LIN {X 0,Y 311.51,Z 741.802,A -85,B 0,C 180,E1 -15908.491,E2 -15908.491} C_VEL
LIN {X 0,Y 309.243,Z 751.676,A -85,B 0,C 180,E1 -15910.758,E2 -15910.758} C_VEL
LIN {X 0,Y 307.436,Z 759.867,A -85,B 0,C 180,E1 -15913.052,E2 -15913.052} C_VEL
LIN {X 0,Y 306.027,Z 766.633,A -85,B 0,C 180,E1 -15915.366,E2 -15915.366} C_VEL
LIN {X 0,Y 304.868,Z 772.893,A -85,B 0,C 180,E1 -15918.024,E2 -15918.024} C_VEL
LIN {X 0,Y 304.197,Z 777.728,A -85,B 0,C 180,E1 -15920.691,E2 -15920.691} C_VEL
LIN {X 0,Y 303.83,Z 781.267,A -85,B 0,C 180,E1 -15923.357,E2 -15923.357} C_VEL
LIN {X 0,Y 303.672,Z 783.591,A -85,B 0,C 180,E1 -15926.017,E2 -15926.017} C_VEL
LIN {X 0,Y 303.588,Z 784.756,A -85,B 0,C 180,E1 -15928.671,E2 -15928.671} C_VEL
LIN {X 0,Y 303.591,Z 784.754,A -85,B 0,C 180,E1 -15931.324,E2 -15931.324} C_VEL
LIN {X 0,Y 303.669,Z 783.578,A -85,B 0,C 180,E1 -15933.979,E2 -15933.979} C_VEL
LIN {X 0,Y 303.822,Z 781.247,A -85,B 0,C 180,E1 -15936.64,E2 -15936.64} C_VEL
LIN {X 0,Y 304.19,Z 777.706,A -85,B 0,C 180,E1 -15939.305,E2 -15939.305} C_VEL
LIN {X 0,Y 304.86,Z 772.864,A -85,B 0,C 180,E1 -15941.972,E2 -15941.972} C_VEL
LIN {X 0,Y 306.013,Z 766.587,A -85,B 0,C 180,E1 -15944.631,E2 -15944.631} C_VEL
LIN {X 0,Y 307.395,Z 759.808,A -85,B 0,C 180,E1 -15946.946,E2 -15946.946} C_VEL
LIN {X 0,Y 309.187,Z 751.614,A -85,B 0,C 180,E1 -15949.242,E2 -15949.242} C_VEL
LIN {X 0,Y 311.488,Z 741.725,A -85,B 0,C 180,E1 -15951.506,E2 -15951.506} C_VEL
LIN {X 0,Y 313.665,Z 731.299,A -85,B 0,C 180,E1 -15953.489,E2 -15953.489} C_VEL
LIN {X 0,Y 316.132,Z 719.493,A -85,B 0,C 180,E1 -15955.335,E2 -15955.335} C_VEL
LIN {X 0,Y 318.535,Z 707.338,A -85,B 0,C 180,E1 -15956.889,E2 -15956.889} C_VEL
LIN {X 0,Y 320.812,Z 694.087,A -85,B 0,C 180,E1 -15958.275,E2 -15958.275} C_VEL
LIN {X 0,Y 323.032,Z 679.121,A -85,B 0,C 180,E1 -15959.512,E2 -15959.512} C_VEL
LIN {X 0,Y 324.845,Z 663.83,A -85,B 0,C 180,E1 -15960.466,E2 -15960.466} C_VEL
LIN {X 0,Y 326.219,Z 648.861,A -85,B 0,C 180,E1 -15961.132,E2 -15961.132} C_VEL
LIN {X 0,Y 327.138,Z 633.341,A -85,B 0,C 180,E1 -15961.575,E2 -15961.575} C_VEL
LIN {X 0,Y 330.856,Z 523.52,A -85,B 0,C 180,E1 -15963.945,E2 -15963.945} C_VEL
LIN {X 0,Y 331.141,Z 509.643,A -85,B 0,C 180,E1 -15964.267,E2 -15964.267} C_VEL
LIN {X 0,Y 327.742,Z 479.595,A -85,B 0,C 180,E1 -15965.462,E2 -15965.462} C_VEL
LIN {X 0,Y 326.078,Z 466.092,A -85,B 0,C 180,E1 -15966.07,E2 -15966.07} C_VEL
LIN {X 0,Y 325.805,Z 448.606,A -85,B 0,C 180,E1 -15967.417,E2 -15967.417} C_VEL
LIN {X 0,Y 321.272,Z 435.052,A -85,B 0,C 180,E1 -15969.052,E2 -15969.052} C_VEL
LIN {X 0,Y 313.204,Z 412.88,A -85,B 0,C 180,E1 -15972.111,E2 -15972.111} C_VEL
LIN {X 0,Y 308.058,Z 399.307,A -85,B 0,C 180,E1 -15974.234,E2 -15974.234} C_VEL
LIN {X 0,Y 305.54,Z 393.805,A -85,B 0,C 180,E1 -15975.294,E2 -15975.294} C_VEL
LIN {X 0,Y 305.42,Z 393.142,A -85,B 0,C 180,E1 -15975.621,E2 -15975.621} C_VEL
LIN {X 0,Y 305.397,Z 393.032,A -85,B 0,C 180,E1 -15979.409,E2 -15979.409} C_VEL
LIN {X 0,Y 305.44,Z 393.013,A -85,B 0,C 180,E1 -15983.256,E2 -15983.256} C_VEL
LIN {X 0,Y 305.451,Z 393.016,A -85,B 0,C 180,E1 -15986.482,E2 -15986.482} C_VEL
LIN {X 0,Y 305.404,Z 393.06,A -85,B 0,C 180,E1 -15989.585,E2 -15989.585} C_VEL
LIN {X 0,Y 305.436,Z 393.062,A -85,B 0,C 180,E1 -15992.6,E2 -15992.6} C_VEL
LIN {X 0,Y 305.426,Z 393.045,A -85,B 0,C 180,E1 -15995.532,E2 -15995.532} C_VEL
LIN {X 0,Y 305.465,Z 393.04,A -85,B 0,C 180,E1 -15999.811,E2 -15999.811} C_VEL
LIN {X 0,Y 305.498,Z 393.042,A -85,B 0,C 180,E1 -16003.975,E2 -16003.975} C_VEL
LIN {X 0,Y 305.556,Z 393.039,A -85,B 0,C 180,E1 -16006.703,E2 -16006.703} C_VEL
LIN {X 0,Y 305.738,Z 393.007,A -85,B 0,C 180,E1 -16011.262,E2 -16011.262} C_VEL
LIN {X 0,Y 305.768,Z 393.02,A -85,B 0,C 180,E1 -16013.401,E2 -16013.401} C_VEL
LIN {X 0,Y 305.842,Z 393.002,A -85,B 0,C 180,E1 -16017.366,E2 -16017.366} C_VEL
LIN {X 0,Y 305.897,Z 392.991,A -85,B 0,C 180,E1 -16020,E2 -16020} C_VEL
LIN {X 0,Y 305.841,Z 393,A -85,B 0,C 180,E1 -16022.634,E2 -16022.634} C_VEL
LIN {X 0,Y 305.778,Z 392.998,A -85,B 0,C 180,E1 -16026.659,E2 -16026.659} C_VEL
LIN {X 0,Y 305.68,Z 393.031,A -85,B 0,C 180,E1 -16029.262,E2 -16029.262} C_VEL
LIN {X 0,Y 305.571,Z 393.035,A -85,B 0,C 180,E1 -16033.297,E2 -16033.297} C_VEL
LIN {X 0,Y 305.536,Z 393.032,A -85,B 0,C 180,E1 -16036.023,E2 -16036.023} C_VEL
LIN {X 0,Y 305.469,Z 393.047,A -85,B 0,C 180,E1 -16040.189,E2 -16040.189} C_VEL
LIN {X 0,Y 305.441,Z 393.053,A -85,B 0,C 180,E1 -16044.467,E2 -16044.467} C_VEL
LIN {X 0,Y 305.427,Z 393.066,A -85,B 0,C 180,E1 -16047.401,E2 -16047.401} C_VEL
LIN {X 0,Y 305.402,Z 393.064,A -85,B 0,C 180,E1 -16050.416,E2 -16050.416} C_VEL
LIN {X 0,Y 305.452,Z 393.063,A -85,B 0,C 180,E1 -16054.08,E2 -16054.08} C_VEL
LIN {X 0,Y 305.482,Z 393.203,A -85,B 0,C 180,E1 -16057.358,E2 -16057.358} C_VEL
LIN {X 0,Y 305.741,Z 394.316,A -85,B 0,C 180,E1 -16057.736,E2 -16057.736} C_VEL
LIN {X 0,Y 309.903,Z 403.344,A -85,B 0,C 180,E1 -16060.265,E2 -16060.265} C_VEL
LIN {X 0,Y 314.349,Z 413.937,A -85,B 0,C 180,E1 -16062.992,E2 -16062.992} C_VEL
LIN {X 0,Y 318.731,Z 425.827,A -85,B 0,C 180,E1 -16065.777,E2 -16065.777} C_VEL
LIN {X 0,Y 323.124,Z 439.562,A -85,B 0,C 180,E1 -16068.69,E2 -16068.69} C_VEL
LIN {X 0,Y 326.921,Z 453.659,A -85,B 0,C 180,E1 -16071.436,E2 -16071.436} C_VEL
LIN {X 0,Y 326.873,Z 456.261,A -85,B 0,C 180,E1 -16071.822,E2 -16071.822} C_VEL
LIN {X 0,Y 325.43,Z 471.142,A -85,B 0,C 180,E1 -16073.782,E2 -16073.782} C_VEL
LIN {X 0,Y 330.701,Z 506.455,A -85,B 0,C 180,E1 -16075.375,E2 -16075.375} C_VEL
LIN {X 0,Y 331.832,Z 515.303,A -85,B 0,C 180,E1 -16075.737,E2 -16075.737} C_VEL
LIN {X 0,Y 327.343,Z 640.026,A -85,B 0,C 180,E1 -16078.447,E2 -16078.447} C_VEL
LIN {X 0,Y 326.311,Z 654.854,A -85,B 0,C 180,E1 -16078.968,E2 -16078.968} C_VEL
LIN {X 0,Y 324.755,Z 669.473,A -85,B 0,C 180,E1 -16079.704,E2 -16079.704} C_VEL
LIN {X 0,Y 323.032,Z 683.041,A -85,B 0,C 180,E1 -16080.627,E2 -16080.627} C_VEL
LIN {X 0,Y 321.047,Z 696.083,A -85,B 0,C 180,E1 -16081.748,E2 -16081.748} C_VEL
LIN {X 0,Y 318.679,Z 709.073,A -85,B 0,C 180,E1 -16083.124,E2 -16083.124} C_VEL
LIN {X 0,Y 316.289,Z 721.052,A -85,B 0,C 180,E1 -16084.678,E2 -16084.678} C_VEL
LIN {X 0,Y 313.921,Z 732.354,A -85,B 0,C 180,E1 -16086.461,E2 -16086.461} C_VEL
LIN {X 0,Y 311.612,Z 743.054,A -85,B 0,C 180,E1 -16088.503,E2 -16088.503} C_VEL
LIN {X 0,Y 309.303,Z 752.871,A -85,B 0,C 180,E1 -16090.766,E2 -16090.766} C_VEL
LIN {X 0,Y 307.451,Z 761.017,A -85,B 0,C 180,E1 -16093.058,E2 -16093.058} C_VEL
LIN {X 0,Y 306.102,Z 767.766,A -85,B 0,C 180,E1 -16095.373,E2 -16095.373} C_VEL
LIN {X 0,Y 304.867,Z 774.023,A -85,B 0,C 180,E1 -16098.028,E2 -16098.028} C_VEL
LIN {X 0,Y 304.166,Z 778.858,A -85,B 0,C 180,E1 -16100.694,E2 -16100.694} C_VEL
LIN {X 0,Y 303.721,Z 782.401,A -85,B 0,C 180,E1 -16103.358,E2 -16103.358} C_VEL
LIN {X 0,Y 303.569,Z 784.742,A -85,B 0,C 180,E1 -16106.019,E2 -16106.019} C_VEL
LIN {X 0,Y 303.524,Z 785.934,A -85,B 0,C 180,E1 -16108.675,E2 -16108.675} C_VEL
LIN {X 0,Y 303.524,Z 785.947,A -85,B 0,C 180,E1 -16111.329,E2 -16111.329} C_VEL
LIN {X 0,Y 303.573,Z 784.809,A -85,B 0,C 180,E1 -16113.985,E2 -16113.985} C_VEL
LIN {X 0,Y 303.727,Z 782.518,A -85,B 0,C 180,E1 -16116.646,E2 -16116.646} C_VEL
LIN {X 0,Y 304.163,Z 779.022,A -85,B 0,C 180,E1 -16119.31,E2 -16119.31} C_VEL
LIN {X 0,Y 304.843,Z 774.239,A -85,B 0,C 180,E1 -16121.977,E2 -16121.977} C_VEL
LIN {X 0,Y 306.062,Z 768.049,A -85,B 0,C 180,E1 -16124.633,E2 -16124.633} C_VEL
LIN {X 0,Y 307.413,Z 761.363,A -85,B 0,C 180,E1 -16126.949,E2 -16126.949} C_VEL
LIN {X 0,Y 309.232,Z 753.258,A -85,B 0,C 180,E1 -16129.243,E2 -16129.243} C_VEL
LIN {X 0,Y 311.524,Z 743.522,A -85,B 0,C 180,E1 -16131.508,E2 -16131.508} C_VEL
LIN {X 0,Y 313.77,Z 733.148,A -85,B 0,C 180,E1 -16133.507,E2 -16133.507} C_VEL
LIN {X 0,Y 316.209,Z 721.687,A -85,B 0,C 180,E1 -16135.333,E2 -16135.333} C_VEL
LIN {X 0,Y 318.557,Z 709.84,A -85,B 0,C 180,E1 -16136.891,E2 -16136.891} C_VEL
LIN {X 0,Y 320.91,Z 697.03,A -85,B 0,C 180,E1 -16138.269,E2 -16138.269} C_VEL
LIN {X 0,Y 323.052,Z 683.358,A -85,B 0,C 180,E1 -16139.455,E2 -16139.455} C_VEL
LIN {X 0,Y 324.751,Z 669.726,A -85,B 0,C 180,E1 -16140.39,E2 -16140.39} C_VEL
LIN {X 0,Y 326.411,Z 654.339,A -85,B 0,C 180,E1 -16141.161,E2 -16141.161} C_VEL
LIN {X 0,Y 327.456,Z 639.227,A -85,B 0,C 180,E1 -16141.681,E2 -16141.681} C_VEL
LIN {X 0,Y 329.462,Z 585.341,A -85,B 0,C 180,E1 -16142.858,E2 -16142.858} C_VEL
LIN {X 0,Y 329.075,Z 579.542,A -85,B 0,C 180,E1 -16143.049,E2 -16143.049} C_VEL
LIN {X 0,Y 324.931,Z 560.924,A -85,B 0,C 180,E1 -16144.008,E2 -16144.008} C_VEL
LIN {X 0,Y 324.64,Z 555.123,A -85,B 0,C 180,E1 -16144.195,E2 -16144.195} C_VEL
LIN {X 0,Y 325.935,Z 515.278,A -85,B 0,C 180,E1 -16145.087,E2 -16145.087} C_VEL
LIN {X 0,Y 321.648,Z 484.966,A -85,B 0,C 180,E1 -16146.443,E2 -16146.443} C_VEL
LIN {X 0,Y 319.509,Z 470.657,A -85,B 0,C 180,E1 -16147.15,E2 -16147.15} C_VEL
LIN {X 0,Y 320.884,Z 457.021,A -85,B 0,C 180,E1 -16148.996,E2 -16148.996} C_VEL
LIN {X 0,Y 317.11,Z 442.56,A -85,B 0,C 180,E1 -16151.844,E2 -16151.844} C_VEL
LIN {X 0,Y 312.874,Z 429.099,A -85,B 0,C 180,E1 -16154.812,E2 -16154.812} C_VEL
LIN {X 0,Y 307.95,Z 415.892,A -85,B 0,C 180,E1 -16157.978,E2 -16157.978} C_VEL
LIN {X 0,Y 303.696,Z 405.879,A -85,B 0,C 180,E1 -16160.639,E2 -16160.639} C_VEL
LIN {X 0,Y 300.029,Z 397.65,A -85,B 0,C 180,E1 -16163.014,E2 -16163.014} C_VEL
LIN {X 0,Y 298.526,Z 394.473,A -85,B 0,C 180,E1 -16163.997,E2 -16163.997} C_VEL
LIN {X 0,Y 298.417,Z 394.003,A -85,B 0,C 180,E1 -16164.346,E2 -16164.346} C_VEL
LIN {X 0,Y 298.392,Z 393.94,A -85,B 0,C 180,E1 -16167.987,E2 -16167.987} C_VEL
LIN {X 0,Y 298.484,Z 394.192,A -85,B 0,C 180,E1 -16169.537,E2 -16169.537} C_VEL
LIN {X 0,Y 298.998,Z 396.184,A -85,B 0,C 180,E1 -16170.007,E2 -16170.007} C_VEL
LIN {X 0,Y 312.309,Z 431.145,A -85,B 0,C 180,E1 -16172.236,E2 -16172.236} C_VEL
LIN {X 0,Y 307.592,Z 539.311,A -85,B 0,C 180,E1 -16175.806,E2 -16175.806} C_VEL
LIN {X 0,Y 307.066,Z 554.35,A -85,B 0,C 180,E1 -16176.519,E2 -16176.519} C_VEL
LIN {X 0,Y 306.274,Z 569.25,A -85,B 0,C 180,E1 -16177.485,E2 -16177.485} C_VEL
LIN {X 0,Y 305.198,Z 584.24,A -85,B 0,C 180,E1 -16178.735,E2 -16178.735} C_VEL
LIN {X 0,Y 304.163,Z 598.638,A -85,B 0,C 180,E1 -16180.249,E2 -16180.249} C_VEL
LIN {X 0,Y 302.949,Z 611.433,A -85,B 0,C 180,E1 -16181.904,E2 -16181.904} C_VEL
LIN {X 0,Y 301.951,Z 623.38,A -85,B 0,C 180,E1 -16183.781,E2 -16183.781} C_VEL
LIN {X 0,Y 300.907,Z 634.09,A -85,B 0,C 180,E1 -16185.804,E2 -16185.804} C_VEL
LIN {X 0,Y 300.192,Z 643.06,A -85,B 0,C 180,E1 -16187.836,E2 -16187.836} C_VEL
LIN {X 0,Y 299.586,Z 650.819,A -85,B 0,C 180,E1 -16189.935,E2 -16189.935} C_VEL
LIN {X 0,Y 299.197,Z 656.877,A -85,B 0,C 180,E1 -16191.898,E2 -16191.898} C_VEL
LIN {X 0,Y 298.839,Z 662.121,A -85,B 0,C 180,E1 -16193.925,E2 -16193.925} C_VEL
LIN {X 0,Y 298.663,Z 666.427,A -85,B 0,C 180,E1 -16195.952,E2 -16195.952} C_VEL
LIN {X 0,Y 298.847,Z 670.682,A -85,B 0,C 180,E1 -16198.652,E2 -16198.652} C_VEL
LIN {X 0,Y 298.852,Z 672.272,A -85,B 0,C 180,E1 -16200,E2 -16200} C_VEL
LIN {X 0,Y 299.267,Z 673.462,A -85,B 0,C 180,E1 -16201.346,E2 -16201.346} C_VEL
LIN {X 0,Y 300.003,Z 674.835,A -85,B 0,C 180,E1 -16204.03,E2 -16204.03} C_VEL
LIN {X 0,Y 300.948,Z 674.817,A -85,B 0,C 180,E1 -16206.705,E2 -16206.705} C_VEL
LIN {X 0,Y 302.425,Z 673.384,A -85,B 0,C 180,E1 -16209.362,E2 -16209.362} C_VEL
LIN {X 0,Y 304.218,Z 670.531,A -85,B 0,C 180,E1 -16212,E2 -16212} C_VEL
LIN {X 0,Y 306.592,Z 666.12,A -85,B 0,C 180,E1 -16214.605,E2 -16214.605} C_VEL
LIN {X 0,Y 309.31,Z 660.084,A -85,B 0,C 180,E1 -16217.18,E2 -16217.18} C_VEL
LIN {X 0,Y 312.514,Z 652.305,A -85,B 0,C 180,E1 -16219.714,E2 -16219.714} C_VEL
LIN {X 0,Y 315.653,Z 643.731,A -85,B 0,C 180,E1 -16221.897,E2 -16221.897} C_VEL
LIN {X 0,Y 319.213,Z 633.249,A -85,B 0,C 180,E1 -16224.036,E2 -16224.036} C_VEL
LIN {X 0,Y 322.424,Z 622.399,A -85,B 0,C 180,E1 -16225.845,E2 -16225.845} C_VEL
LIN {X 0,Y 325.632,Z 610.523,A -85,B 0,C 180,E1 -16227.473,E2 -16227.473} C_VEL
LIN {X 0,Y 328.416,Z 598.92,A -85,B 0,C 180,E1 -16228.782,E2 -16228.782} C_VEL
LIN {X 0,Y 331.352,Z 584.909,A -85,B 0,C 180,E1 -16230.072,E2 -16230.072} C_VEL
LIN {X 0,Y 333.715,Z 571.514,A -85,B 0,C 180,E1 -16231.062,E2 -16231.062} C_VEL
LIN {X 0,Y 335.94,Z 555.723,A -85,B 0,C 180,E1 -16231.975,E2 -16231.975} C_VEL
LIN {X 0,Y 339.552,Z 531.528,A -85,B 0,C 180,E1 -16233.086,E2 -16233.086} C_VEL
LIN {X 0,Y 350.202,Z 471.926,A -85,B 0,C 180,E1 -16235.552,E2 -16235.552} C_VEL
LIN {X 0,Y 348.137,Z 468.686,A -85,B 0,C 180,E1 -16237.052,E2 -16237.052} C_VEL
LIN {X 0,Y 346.664,Z 466.644,A -85,B 0,C 180,E1 -16238.416,E2 -16238.416} C_VEL
LIN {X 0,Y 345.343,Z 465.295,A -85,B 0,C 180,E1 -16240.093,E2 -16240.093} C_VEL
LIN {X 0,Y 344.375,Z 465.546,A -85,B 0,C 180,E1 -16242.335,E2 -16242.335} C_VEL
LIN {X 0,Y 344.393,Z 467.057,A -85,B 0,C 180,E1 -16244.225,E2 -16244.225} C_VEL
LIN {X 0,Y 345.076,Z 469.965,A -85,B 0,C 180,E1 -16246.041,E2 -16246.041} C_VEL
LIN {X 0,Y 346.193,Z 473.917,A -85,B 0,C 180,E1 -16247.668,E2 -16247.668} C_VEL
LIN {X 0,Y 347.072,Z 477.937,A -85,B 0,C 180,E1 -16248.757,E2 -16248.757} C_VEL
LIN {X 0,Y 346.126,Z 493.091,A -85,B 0,C 180,E1 -16250.169,E2 -16250.169} C_VEL
LIN {X 0,Y 345.134,Z 507.077,A -85,B 0,C 180,E1 -16251.23,E2 -16251.23} C_VEL
LIN {X 0,Y 344.11,Z 517.462,A -85,B 0,C 180,E1 -16251.846,E2 -16251.846} C_VEL
LIN {X 0,Y 334.494,Z 583.589,A -85,B 0,C 180,E1 -16254.333,E2 -16254.333} C_VEL
LIN {X 0,Y 331.162,Z 606.428,A -85,B 0,C 180,E1 -16255.224,E2 -16255.224} C_VEL
LIN {X 0,Y 327.559,Z 624.762,A -85,B 0,C 180,E1 -16256.184,E2 -16256.184} C_VEL
LIN {X 0,Y 323.528,Z 641.309,A -85,B 0,C 180,E1 -16257.29,E2 -16257.29} C_VEL
LIN {X 0,Y 319.664,Z 655.712,A -85,B 0,C 180,E1 -16258.475,E2 -16258.475} C_VEL
LIN {X 0,Y 318.027,Z 670.659,A -85,B 0,C 180,E1 -16259.265,E2 -16259.265} C_VEL
LIN {X 0,Y 316.199,Z 684.903,A -85,B 0,C 180,E1 -16260.295,E2 -16260.295} C_VEL
LIN {X 0,Y 313.837,Z 698.991,A -85,B 0,C 180,E1 -16261.582,E2 -16261.582} C_VEL
LIN {X 0,Y 311.474,Z 711.335,A -85,B 0,C 180,E1 -16262.991,E2 -16262.991} C_VEL
LIN {X 0,Y 308.815,Z 723.869,A -85,B 0,C 180,E1 -16264.739,E2 -16264.739} C_VEL
LIN {X 0,Y 306.436,Z 734.513,A -85,B 0,C 180,E1 -16266.547,E2 -16266.547} C_VEL
LIN {X 0,Y 304.115,Z 744.788,A -85,B 0,C 180,E1 -16268.653,E2 -16268.653} C_VEL
LIN {X 0,Y 301.922,Z 754.151,A -85,B 0,C 180,E1 -16270.979,E2 -16270.979} C_VEL
LIN {X 0,Y 300.11,Z 761.927,A -85,B 0,C 180,E1 -16273.327,E2 -16273.327} C_VEL
LIN {X 0,Y 298.803,Z 768.365,A -85,B 0,C 180,E1 -16275.7,E2 -16275.7} C_VEL
LIN {X 0,Y 297.647,Z 774.26,A -85,B 0,C 180,E1 -16278.42,E2 -16278.42} C_VEL
LIN {X 0,Y 297.163,Z 777.744,A -85,B 0,C 180,E1 -16280.469,E2 -16280.469} C_VEL
LIN {X 0,Y 296.743,Z 781.282,A -85,B 0,C 180,E1 -16283.197,E2 -16283.197} C_VEL
LIN {X 0,Y 296.569,Z 783.605,A -85,B 0,C 180,E1 -16285.921,E2 -16285.921} C_VEL
LIN {X 0,Y 296.508,Z 784.77,A -85,B 0,C 180,E1 -16288.64,E2 -16288.64} C_VEL
LIN {X 0,Y 296.51,Z 784.767,A -85,B 0,C 180,E1 -16291.356,E2 -16291.356} C_VEL
LIN {X 0,Y 296.566,Z 783.592,A -85,B 0,C 180,E1 -16294.075,E2 -16294.075} C_VEL
LIN {X 0,Y 296.736,Z 781.26,A -85,B 0,C 180,E1 -16296.799,E2 -16296.799} C_VEL
LIN {X 0,Y 297.157,Z 777.72,A -85,B 0,C 180,E1 -16299.527,E2 -16299.527} C_VEL
LIN {X 0,Y 297.875,Z 772.878,A -85,B 0,C 180,E1 -16302.257,E2 -16302.257} C_VEL
LIN {X 0,Y 299.095,Z 766.602,A -85,B 0,C 180,E1 -16304.977,E2 -16304.977} C_VEL
LIN {X 0,Y 300.812,Z 758.713,A -85,B 0,C 180,E1 -16307.679,E2 -16307.679} C_VEL
LIN {X 0,Y 302.756,Z 750.291,A -85,B 0,C 180,E1 -16310.021,E2 -16310.021} C_VEL
LIN {X 0,Y 304.85,Z 741.742,A -85,B 0,C 180,E1 -16311.999,E2 -16311.999} C_VEL
LIN {X 0,Y 307.091,Z 731.493,A -85,B 0,C 180,E1 -16313.987,E2 -16313.987} C_VEL
LIN {X 0,Y 309.731,Z 719.513,A -85,B 0,C 180,E1 -16315.897,E2 -16315.897} C_VEL
LIN {X 0,Y 312.201,Z 707.36,A -85,B 0,C 180,E1 -16317.48,E2 -16317.48} C_VEL
LIN {X 0,Y 314.56,Z 694.113,A -85,B 0,C 180,E1 -16318.889,E2 -16318.889} C_VEL
LIN {X 0,Y 316.743,Z 680.031,A -85,B 0,C 180,E1 -16320.078,E2 -16320.078} C_VEL
LIN {X 0,Y 318.589,Z 665.264,A -85,B 0,C 180,E1 -16321.038,E2 -16321.038} C_VEL
LIN {X 0,Y 320.103,Z 649.948,A -85,B 0,C 180,E1 -16321.749,E2 -16321.749} C_VEL
LIN {X 0,Y 321.029,Z 635.079,A -85,B 0,C 180,E1 -16322.201,E2 -16322.201} C_VEL
LIN {X 0,Y 324.415,Z 540.245,A -85,B 0,C 180,E1 -16324.278,E2 -16324.278} C_VEL
LIN {X 0,Y 325.335,Z 511.034,A -85,B 0,C 180,E1 -16324.933,E2 -16324.933} C_VEL
LIN {X 0,Y 321.895,Z 480.308,A -85,B 0,C 180,E1 -16326.19,E2 -16326.19} C_VEL
LIN {X 0,Y 320.242,Z 466.176,A -85,B 0,C 180,E1 -16326.835,E2 -16326.835} C_VEL
LIN {X 0,Y 319.986,Z 450.746,A -85,B 0,C 180,E1 -16328.077,E2 -16328.077} C_VEL
LIN {X 0,Y 315.058,Z 436.228,A -85,B 0,C 180,E1 -16329.947,E2 -16329.947} C_VEL
LIN {X 0,Y 311.413,Z 425.92,A -85,B 0,C 180,E1 -16331.376,E2 -16331.376} C_VEL
LIN {X 0,Y 307.502,Z 414.909,A -85,B 0,C 180,E1 -16332.999,E2 -16332.999} C_VEL
LIN {X 0,Y 303.233,Z 403.406,A -85,B 0,C 180,E1 -16334.838,E2 -16334.838} C_VEL
LIN {X 0,Y 300.526,Z 398.196,A -85,B 0,C 180,E1 -16335.916,E2 -16335.916} C_VEL
LIN {X 0,Y 298.846,Z 395.687,A -85,B 0,C 180,E1 -16336.539,E2 -16336.539} C_VEL
LIN {X 0,Y 298.422,Z 394.203,A -85,B 0,C 180,E1 -16336.924,E2 -16336.924} C_VEL
LIN {X 0,Y 298.358,Z 393.893,A -85,B 0,C 180,E1 -16337.83,E2 -16337.83} C_VEL
LIN {X 0,Y 298.385,Z 393.913,A -85,B 0,C 180,E1 -16342.238,E2 -16342.238} C_VEL
LIN {X 0,Y 298.394,Z 393.88,A -85,B 0,C 180,E1 -16345.579,E2 -16345.579} C_VEL
LIN {X 0,Y 298.36,Z 393.946,A -85,B 0,C 180,E1 -16348.787,E2 -16348.787} C_VEL
LIN {X 0,Y 298.39,Z 393.931,A -85,B 0,C 180,E1 -16351.897,E2 -16351.897} C_VEL
LIN {X 0,Y 298.4,Z 393.921,A -85,B 0,C 180,E1 -16354.916,E2 -16354.916} C_VEL
LIN {X 0,Y 298.378,Z 393.944,A -85,B 0,C 180,E1 -16357.861,E2 -16357.861} C_VEL
LIN {X 0,Y 298.445,Z 393.916,A -85,B 0,C 180,E1 -16360.751,E2 -16360.751} C_VEL
LIN {X 0,Y 298.496,Z 393.905,A -85,B 0,C 180,E1 -16364.99,E2 -16364.99} C_VEL
LIN {X 0,Y 298.567,Z 393.905,A -85,B 0,C 180,E1 -16369.146,E2 -16369.146} C_VEL
LIN {X 0,Y 298.681,Z 393.893,A -85,B 0,C 180,E1 -16371.884,E2 -16371.884} C_VEL
LIN {X 0,Y 298.613,Z 393.896,A -85,B 0,C 180,E1 -16374.598,E2 -16374.598} C_VEL
LIN {X 0,Y 298.888,Z 393.88,A -85,B 0,C 180,E1 -16378.653,E2 -16378.653} C_VEL
LIN {X 0,Y 298.899,Z 393.854,A -85,B 0,C 180,E1 -16381.347,E2 -16381.347} C_VEL
LIN {X 0,Y 298.732,Z 393.876,A -85,B 0,C 180,E1 -16386.756,E2 -16386.756} C_VEL
LIN {X 0,Y 298.611,Z 393.911,A -85,B 0,C 180,E1 -16389.483,E2 -16389.483} C_VEL
LIN {X 0,Y 298.53,Z 393.918,A -85,B 0,C 180,E1 -16393.617,E2 -16393.617} C_VEL
LIN {X 0,Y 298.469,Z 393.91,A -85,B 0,C 180,E1 -16396.413,E2 -16396.413} C_VEL
LIN {X 0,Y 298.428,Z 393.931,A -85,B 0,C 180,E1 -16399.618,E2 -16399.618} C_VEL
LIN {X 0,Y 298.375,Z 393.943,A -85,B 0,C 180,E1 -16403.605,E2 -16403.605} C_VEL
LIN {X 0,Y 298.388,Z 393.933,A -85,B 0,C 180,E1 -16406.584,E2 -16406.584} C_VEL
LIN {X 0,Y 298.343,Z 393.936,A -85,B 0,C 180,E1 -16409.65,E2 -16409.65} C_VEL
LIN {X 0,Y 298.38,Z 393.934,A -85,B 0,C 180,E1 -16412.802,E2 -16412.802} C_VEL
LIN {X 0,Y 298.447,Z 394.152,A -85,B 0,C 180,E1 -16416.014,E2 -16416.014} C_VEL
LIN {X 0,Y 299.785,Z 397.321,A -85,B 0,C 180,E1 -16417.021,E2 -16417.021} C_VEL
LIN {X 0,Y 305.487,Z 409.902,A -85,B 0,C 180,E1 -16420.611,E2 -16420.611} C_VEL
LIN {X 0,Y 310.009,Z 421.278,A -85,B 0,C 180,E1 -16423.498,E2 -16423.498} C_VEL
LIN {X 0,Y 313.539,Z 431.257,A -85,B 0,C 180,E1 -16425.831,E2 -16425.831} C_VEL
LIN {X 0,Y 317.332,Z 443.459,A -85,B 0,C 180,E1 -16428.457,E2 -16428.457} C_VEL
LIN {X 0,Y 320.771,Z 456.424,A -85,B 0,C 180,E1 -16431.017,E2 -16431.017} C_VEL
LIN {X 0,Y 320.123,Z 463.961,A -85,B 0,C 180,E1 -16432.072,E2 -16432.072} C_VEL
LIN {X 0,Y 319.486,Z 471.032,A -85,B 0,C 180,E1 -16432.997,E2 -16432.997} C_VEL
LIN {X 0,Y 324.864,Z 507.58,A -85,B 0,C 180,E1 -16434.694,E2 -16434.694} C_VEL
LIN {X 0,Y 325.887,Z 515.693,A -85,B 0,C 180,E1 -16435.035,E2 -16435.035} C_VEL
LIN {X 0,Y 322.195,Z 618.134,A -85,B 0,C 180,E1 -16437.282,E2 -16437.282} C_VEL
LIN {X 0,Y 321.19,Z 642.694,A -85,B 0,C 180,E1 -16437.863,E2 -16437.863} C_VEL
LIN {X 0,Y 319.938,Z 658.269,A -85,B 0,C 180,E1 -16438.463,E2 -16438.463} C_VEL
LIN {X 0,Y 318.201,Z 673.182,A -85,B 0,C 180,E1 -16439.289,E2 -16439.289} C_VEL
LIN {X 0,Y 316.214,Z 687.227,A -85,B 0,C 180,E1 -16440.331,E2 -16440.331} C_VEL
LIN {X 0,Y 313.951,Z 700.694,A -85,B 0,C 180,E1 -16441.598,E2 -16441.598} C_VEL
LIN {X 0,Y 311.282,Z 714.117,A -85,B 0,C 180,E1 -16443.159,E2 -16443.159} C_VEL
LIN {X 0,Y 308.717,Z 726.285,A -85,B 0,C 180,E1 -16444.915,E2 -16444.915} C_VEL
LIN {X 0,Y 306.509,Z 736.36,A -85,B 0,C 180,E1 -16446.675,E2 -16446.675} C_VEL
LIN {X 0,Y 304.19,Z 745.986,A -85,B 0,C 180,E1 -16448.663,E2 -16448.663} C_VEL
LIN {X 0,Y 301.966,Z 755.297,A -85,B 0,C 180,E1 -16450.986,E2 -16450.986} C_VEL
LIN {X 0,Y 300.356,Z 762.046,A -85,B 0,C 180,E1 -16452.996,E2 -16452.996} C_VEL
LIN {X 0,Y 298.857,Z 769.471,A -85,B 0,C 180,E1 -16455.707,E2 -16455.707} C_VEL
LIN {X 0,Y 297.641,Z 775.367,A -85,B 0,C 180,E1 -16458.424,E2 -16458.424} C_VEL
LIN {X 0,Y 297.107,Z 778.845,A -85,B 0,C 180,E1 -16460.471,E2 -16460.471} C_VEL
LIN {X 0,Y 296.645,Z 782.388,A -85,B 0,C 180,E1 -16463.199,E2 -16463.199} C_VEL
LIN {X 0,Y 296.47,Z 784.729,A -85,B 0,C 180,E1 -16465.924,E2 -16465.924} C_VEL
LIN {X 0,Y 296.445,Z 785.92,A -85,B 0,C 180,E1 -16468.644,E2 -16468.644} C_VEL
LIN {X 0,Y 296.446,Z 785.933,A -85,B 0,C 180,E1 -16471.361,E2 -16471.361} C_VEL
LIN {X 0,Y 296.476,Z 784.794,A -85,B 0,C 180,E1 -16474.08,E2 -16474.08} C_VEL
LIN {X 0,Y 296.65,Z 782.503,A -85,B 0,C 180,E1 -16476.805,E2 -16476.805} C_VEL
LIN {X 0,Y 297.102,Z 779.006,A -85,B 0,C 180,E1 -16479.533,E2 -16479.533} C_VEL
LIN {X 0,Y 297.862,Z 774.223,A -85,B 0,C 180,E1 -16482.262,E2 -16482.262} C_VEL
LIN {X 0,Y 299.152,Z 768.031,A -85,B 0,C 180,E1 -16484.979,E2 -16484.979} C_VEL
LIN {X 0,Y 300.827,Z 760.243,A -85,B 0,C 180,E1 -16487.682,E2 -16487.682} C_VEL
LIN {X 0,Y 302.756,Z 751.933,A -85,B 0,C 180,E1 -16490.025,E2 -16490.025} C_VEL
LIN {X 0,Y 305.21,Z 741.924,A -85,B 0,C 180,E1 -16492.332,E2 -16492.332} C_VEL
LIN {X 0,Y 307.513,Z 731.7,A -85,B 0,C 180,E1 -16494.293,E2 -16494.293} C_VEL
LIN {X 0,Y 310.051,Z 720.594,A -85,B 0,C 180,E1 -16496.053,E2 -16496.053} C_VEL
LIN {X 0,Y 312.459,Z 708.544,A -85,B 0,C 180,E1 -16497.641,E2 -16497.641} C_VEL
LIN {X 0,Y 314.958,Z 695.45,A -85,B 0,C 180,E1 -16499.036,E2 -16499.036} C_VEL
LIN {X 0,Y 317.212,Z 681.03,A -85,B 0,C 180,E1 -16500.27,E2 -16500.27} C_VEL
LIN {X 0,Y 318.959,Z 667.168,A -85,B 0,C 180,E1 -16501.187,E2 -16501.187} C_VEL
LIN {X 0,Y 320.582,Z 651.666,A -85,B 0,C 180,E1 -16501.932,E2 -16501.932} C_VEL
LIN {X 0,Y 321.568,Z 636.362,A -85,B 0,C 180,E1 -16502.423,E2 -16502.423} C_VEL
LIN {X 0,Y 324.64,Z 555.123,A -85,B 0,C 180,E1 -16504.195,E2 -16504.195} C_VEL
LIN {X 0,Y 324.323,Z 549.324,A -85,B 0,C 180,E1 -16504.385,E2 -16504.385} C_VEL
LIN {X 0,Y 320.15,Z 530.757,A -85,B 0,C 180,E1 -16505.395,E2 -16505.395} C_VEL
LIN {X 0,Y 319.861,Z 524.957,A -85,B 0,C 180,E1 -16505.588,E2 -16505.588} C_VEL
LIN {X 0,Y 320.086,Z 516.087,A -85,B 0,C 180,E1 -16505.8,E2 -16505.8} C_VEL
LIN {X 0,Y 315.942,Z 486.343,A -85,B 0,C 180,E1 -16507.167,E2 -16507.167} C_VEL
LIN {X 0,Y 313.602,Z 470.582,A -85,B 0,C 180,E1 -16507.971,E2 -16507.971} C_VEL
LIN {X 0,Y 314.724,Z 460.401,A -85,B 0,C 180,E1 -16509.333,E2 -16509.333} C_VEL
LIN {X 0,Y 312.386,Z 450.248,A -85,B 0,C 180,E1 -16511.331,E2 -16511.331} C_VEL
LIN {X 0,Y 308.544,Z 437.135,A -85,B 0,C 180,E1 -16514.151,E2 -16514.151} C_VEL
LIN {X 0,Y 303.777,Z 423.484,A -85,B 0,C 180,E1 -16517.413,E2 -16517.413} C_VEL
LIN {X 0,Y 298.897,Z 411.47,A -85,B 0,C 180,E1 -16520.591,E2 -16520.591} C_VEL
LIN {X 0,Y 293.042,Z 398.611,A -85,B 0,C 180,E1 -16524.438,E2 -16524.438} C_VEL
LIN {X 0,Y 291.422,Z 395.06,A -85,B 0,C 180,E1 -16525.629,E2 -16525.629} C_VEL
LIN {X 0,Y 291.343,Z 394.806,A -85,B 0,C 180,E1 -16527.6,E2 -16527.6} C_VEL
LIN {X 0,Y 291.404,Z 395.022,A -85,B 0,C 180,E1 -16529.069,E2 -16529.069} C_VEL
LIN {X 0,Y 291.863,Z 396.732,A -85,B 0,C 180,E1 -16529.494,E2 -16529.494} C_VEL
LIN {X 0,Y 305.488,Z 432.593,A -85,B 0,C 180,E1 -16531.846,E2 -16531.846} C_VEL
LIN {X 0,Y 300.68,Z 540.479,A -85,B 0,C 180,E1 -16535.515,E2 -16535.515} C_VEL
LIN {X 0,Y 300.14,Z 555.785,A -85,B 0,C 180,E1 -16536.272,E2 -16536.272} C_VEL
LIN {X 0,Y 299.267,Z 570.932,A -85,B 0,C 180,E1 -16537.293,E2 -16537.293} C_VEL
LIN {X 0,Y 298.207,Z 585.717,A -85,B 0,C 180,E1 -16538.574,E2 -16538.574} C_VEL
LIN {X 0,Y 297.089,Z 599.93,A -85,B 0,C 180,E1 -16540.119,E2 -16540.119} C_VEL
LIN {X 0,Y 295.872,Z 612.781,A -85,B 0,C 180,E1 -16541.836,E2 -16541.836} C_VEL
LIN {X 0,Y 294.854,Z 624.554,A -85,B 0,C 180,E1 -16543.736,E2 -16543.736} C_VEL
LIN {X 0,Y 293.83,Z 635.289,A -85,B 0,C 180,E1 -16545.808,E2 -16545.808} C_VEL
LIN {X 0,Y 293.089,Z 644.27,A -85,B 0,C 180,E1 -16547.888,E2 -16547.888} C_VEL
LIN {X 0,Y 292.412,Z 652.958,A -85,B 0,C 180,E1 -16550.314,E2 -16550.314} C_VEL
LIN {X 0,Y 292.107,Z 659.081,A -85,B 0,C 180,E1 -16552.396,E2 -16552.396} C_VEL
LIN {X 0,Y 291.633,Z 664.124,A -85,B 0,C 180,E1 -16554.468,E2 -16554.468} C_VEL
LIN {X 0,Y 291.646,Z 669.42,A -85,B 0,C 180,E1 -16557.237,E2 -16557.237} C_VEL
LIN {X 0,Y 291.817,Z 671.472,A -85,B 0,C 180,E1 -16558.62,E2 -16558.62} C_VEL
LIN {X 0,Y 291.823,Z 673.168,A -85,B 0,C 180,E1 -16560,E2 -16560} C_VEL
LIN {X 0,Y 292.257,Z 674.451,A -85,B 0,C 180,E1 -16561.378,E2 -16561.378} C_VEL
LIN {X 0,Y 293.029,Z 676.01,A -85,B 0,C 180,E1 -16564.126,E2 -16564.126} C_VEL
LIN {X 0,Y 294.039,Z 676.191,A -85,B 0,C 180,E1 -16566.864,E2 -16566.864} C_VEL
LIN {X 0,Y 295.607,Z 674.942,A -85,B 0,C 180,E1 -16569.58,E2 -16569.58} C_VEL
LIN {X 0,Y 297.516,Z 672.32,A -85,B 0,C 180,E1 -16572.275,E2 -16572.275} C_VEL
LIN {X 0,Y 300.031,Z 668.177,A -85,B 0,C 180,E1 -16574.932,E2 -16574.932} C_VEL
LIN {X 0,Y 302.913,Z 662.455,A -85,B 0,C 180,E1 -16577.555,E2 -16577.555} C_VEL
LIN {X 0,Y 305.804,Z 656.105,A -85,B 0,C 180,E1 -16579.78,E2 -16579.78} C_VEL
LIN {X 0,Y 309.111,Z 648.062,A -85,B 0,C 180,E1 -16582.033,E2 -16582.033} C_VEL
LIN {X 0,Y 312.285,Z 639.804,A -85,B 0,C 180,E1 -16583.897,E2 -16583.897} C_VEL
LIN {X 0,Y 315.611,Z 630.066,A -85,B 0,C 180,E1 -16585.736,E2 -16585.736} C_VEL
LIN {X 0,Y 319.193,Z 618.513,A -85,B 0,C 180,E1 -16587.541,E2 -16587.541} C_VEL
LIN {X 0,Y 322.687,Z 605.735,A -85,B 0,C 180,E1 -16589.164,E2 -16589.164} C_VEL
LIN {X 0,Y 326.188,Z 591.531,A -85,B 0,C 180,E1 -16590.598,E2 -16590.598} C_VEL
LIN {X 0,Y 329.01,Z 577.691,A -85,B 0,C 180,E1 -16591.736,E2 -16591.736} C_VEL
LIN {X 0,Y 331.756,Z 561.031,A -85,B 0,C 180,E1 -16592.787,E2 -16592.787} C_VEL
LIN {X 0,Y 334.715,Z 541.954,A -85,B 0,C 180,E1 -16593.718,E2 -16593.718} C_VEL
LIN {X 0,Y 342.511,Z 499.563,A -85,B 0,C 180,E1 -16595.525,E2 -16595.525} C_VEL
LIN {X 0,Y 346.953,Z 477.007,A -85,B 0,C 180,E1 -16596.443,E2 -16596.443} C_VEL
LIN {X 0,Y 345.49,Z 474.65,A -85,B 0,C 180,E1 -16597.681,E2 -16597.681} C_VEL
LIN {X 0,Y 344.538,Z 473.271,A -85,B 0,C 180,E1 -16598.688,E2 -16598.688} C_VEL
LIN {X 0,Y 343.323,Z 472.125,A -85,B 0,C 180,E1 -16600.369,E2 -16600.369} C_VEL
LIN {X 0,Y 342.514,Z 472.574,A -85,B 0,C 180,E1 -16602.619,E2 -16602.619} C_VEL
LIN {X 0,Y 342.634,Z 474.423,A -85,B 0,C 180,E1 -16604.512,E2 -16604.512} C_VEL
LIN {X 0,Y 343.351,Z 477.783,A -85,B 0,C 180,E1 -16606.34,E2 -16606.34} C_VEL
LIN {X 0,Y 343.943,Z 480.319,A -85,B 0,C 180,E1 -16607.292,E2 -16607.292} C_VEL
LIN {X 0,Y 344.345,Z 482.865,A -85,B 0,C 180,E1 -16607.976,E2 -16607.976} C_VEL
LIN {X 0,Y 343.029,Z 497.694,A -85,B 0,C 180,E1 -16609.356,E2 -16609.356} C_VEL
LIN {X 0,Y 341.752,Z 511.035,A -85,B 0,C 180,E1 -16610.353,E2 -16610.353} C_VEL
LIN {X 0,Y 340.821,Z 518.827,A -85,B 0,C 180,E1 -16610.818,E2 -16610.818} C_VEL
LIN {X 0,Y 330.563,Z 584.15,A -85,B 0,C 180,E1 -16613.322,E2 -16613.322} C_VEL
LIN {X 0,Y 327.18,Z 605.34,A -85,B 0,C 180,E1 -16614.171,E2 -16614.171} C_VEL
LIN {X 0,Y 323.667,Z 622.128,A -85,B 0,C 180,E1 -16615.06,E2 -16615.06} C_VEL
LIN {X 0,Y 319.689,Z 637.758,A -85,B 0,C 180,E1 -16616.092,E2 -16616.092} C_VEL
LIN {X 0,Y 314.91,Z 653.909,A -85,B 0,C 180,E1 -16617.423,E2 -16617.423} C_VEL
LIN {X 0,Y 313.233,Z 659.817,A -85,B 0,C 180,E1 -16617.988,E2 -16617.988} C_VEL
LIN {X 0,Y 311.442,Z 674.634,A -85,B 0,C 180,E1 -16618.861,E2 -16618.861} C_VEL
LIN {X 0,Y 309.323,Z 689.202,A -85,B 0,C 180,E1 -16620.008,E2 -16620.008} C_VEL
LIN {X 0,Y 306.731,Z 703.37,A -85,B 0,C 180,E1 -16621.424,E2 -16621.424} C_VEL
LIN {X 0,Y 304.12,Z 716.183,A -85,B 0,C 180,E1 -16623.028,E2 -16623.028} C_VEL
LIN {X 0,Y 301.437,Z 727.899,A -85,B 0,C 180,E1 -16624.816,E2 -16624.816} C_VEL
LIN {X 0,Y 298.977,Z 738.616,A -85,B 0,C 180,E1 -16626.811,E2 -16626.811} C_VEL
LIN {X 0,Y 296.727,Z 747.688,A -85,B 0,C 180,E1 -16628.824,E2 -16628.824} C_VEL
LIN {X 0,Y 294.592,Z 756.572,A -85,B 0,C 180,E1 -16631.21,E2 -16631.21} C_VEL
LIN {X 0,Y 292.618,Z 764.668,A -85,B 0,C 180,E1 -16633.885,E2 -16633.885} C_VEL
LIN {X 0,Y 291.257,Z 771.509,A -85,B 0,C 180,E1 -16636.746,E2 -16636.746} C_VEL
LIN {X 0,Y 290.272,Z 776.698,A -85,B 0,C 180,E1 -16639.536,E2 -16639.536} C_VEL
LIN {X 0,Y 289.87,Z 779.684,A -85,B 0,C 180,E1 -16641.633,E2 -16641.633} C_VEL
LIN {X 0,Y 289.536,Z 782.606,A -85,B 0,C 180,E1 -16644.426,E2 -16644.426} C_VEL
LIN {X 0,Y 289.471,Z 784.344,A -85,B 0,C 180,E1 -16647.215,E2 -16647.215} C_VEL
LIN {X 0,Y 289.427,Z 784.935,A -85,B 0,C 180,E1 -16649.998,E2 -16649.998} C_VEL
LIN {X 0,Y 289.476,Z 784.336,A -85,B 0,C 180,E1 -16652.781,E2 -16652.781} C_VEL
LIN {X 0,Y 289.514,Z 782.587,A -85,B 0,C 180,E1 -16655.57,E2 -16655.57} C_VEL
LIN {X 0,Y 289.842,Z 779.66,A -85,B 0,C 180,E1 -16658.363,E2 -16658.363} C_VEL
LIN {X 0,Y 290.452,Z 775.483,A -85,B 0,C 180,E1 -16661.159,E2 -16661.159} C_VEL
LIN {X 0,Y 291.555,Z 769.943,A -85,B 0,C 180,E1 -16663.946,E2 -16663.946} C_VEL
LIN {X 0,Y 293.016,Z 762.888,A -85,B 0,C 180,E1 -16666.725,E2 -16666.725} C_VEL
LIN {X 0,Y 294.806,Z 755.325,A -85,B 0,C 180,E1 -16669.132,E2 -16669.132} C_VEL
LIN {X 0,Y 297.042,Z 746.206,A -85,B 0,C 180,E1 -16671.511,E2 -16671.511} C_VEL
LIN {X 0,Y 299.274,Z 736.908,A -85,B 0,C 180,E1 -16673.527,E2 -16673.527} C_VEL
LIN {X 0,Y 301.862,Z 725.856,A -85,B 0,C 180,E1 -16675.511,E2 -16675.511} C_VEL
LIN {X 0,Y 304.546,Z 713.731,A -85,B 0,C 180,E1 -16677.298,E2 -16677.298} C_VEL
LIN {X 0,Y 307.272,Z 700.378,A -85,B 0,C 180,E1 -16678.89,E2 -16678.89} C_VEL
LIN {X 0,Y 309.543,Z 687.192,A -85,B 0,C 180,E1 -16680.158,E2 -16680.158} C_VEL
LIN {X 0,Y 311.617,Z 672.857,A -85,B 0,C 180,E1 -16681.244,E2 -16681.244} C_VEL
LIN {X 0,Y 313.339,Z 657.927,A -85,B 0,C 180,E1 -16682.09,E2 -16682.09} C_VEL
LIN {X 0,Y 314.648,Z 642.319,A -85,B 0,C 180,E1 -16682.698,E2 -16682.698} C_VEL
LIN {X 0,Y 316.527,Z 596.175,A -85,B 0,C 180,E1 -16683.755,E2 -16683.755} C_VEL
LIN {X 0,Y 319.578,Z 512.584,A -85,B 0,C 180,E1 -16685.618,E2 -16685.618} C_VEL
LIN {X 0,Y 316.307,Z 482.333,A -85,B 0,C 180,E1 -16686.881,E2 -16686.881} C_VEL
LIN {X 0,Y 314.432,Z 466.261,A -85,B 0,C 180,E1 -16687.632,E2 -16687.632} C_VEL
LIN {X 0,Y 314.342,Z 453.625,A -85,B 0,C 180,E1 -16688.68,E2 -16688.68} C_VEL
LIN {X 0,Y 308.161,Z 434.9,A -85,B 0,C 180,E1 -16691.183,E2 -16691.183} C_VEL
LIN {X 0,Y 302.477,Z 418.694,A -85,B 0,C 180,E1 -16693.629,E2 -16693.629} C_VEL
LIN {X 0,Y 299.095,Z 409.185,A -85,B 0,C 180,E1 -16695.177,E2 -16695.177} C_VEL
LIN {X 0,Y 296.791,Z 404.266,A -85,B 0,C 180,E1 -16696.161,E2 -16696.161} C_VEL
LIN {X 0,Y 293.793,Z 399.312,A -85,B 0,C 180,E1 -16697.349,E2 -16697.349} C_VEL
LIN {X 0,Y 292.649,Z 398.109,A -85,B 0,C 180,E1 -16697.746,E2 -16697.746} C_VEL
LIN {X 0,Y 291.423,Z 395.434,A -85,B 0,C 180,E1 -16698.379,E2 -16698.379} C_VEL
LIN {X 0,Y 291.317,Z 394.799,A -85,B 0,C 180,E1 -16698.86,E2 -16698.86} C_VEL
LIN {X 0,Y 291.377,Z 394.767,A -85,B 0,C 180,E1 -16702.915,E2 -16702.915} C_VEL
LIN {X 0,Y 291.33,Z 394.768,A -85,B 0,C 180,E1 -16706.3,E2 -16706.3} C_VEL
LIN {X 0,Y 291.324,Z 394.806,A -85,B 0,C 180,E1 -16710.276,E2 -16710.276} C_VEL
LIN {X 0,Y 291.329,Z 394.806,A -85,B 0,C 180,E1 -16714.264,E2 -16714.264} C_VEL
LIN {X 0,Y 291.336,Z 394.82,A -85,B 0,C 180,E1 -16717.296,E2 -16717.296} C_VEL
LIN {X 0,Y 291.37,Z 394.795,A -85,B 0,C 180,E1 -16720.264,E2 -16720.264} C_VEL
LIN {X 0,Y 291.46,Z 394.783,A -85,B 0,C 180,E1 -16724.682,E2 -16724.682} C_VEL
LIN {X 0,Y 291.512,Z 394.787,A -85,B 0,C 180,E1 -16728.88,E2 -16728.88} C_VEL
LIN {X 0,Y 291.635,Z 394.767,A -85,B 0,C 180,E1 -16731.687,E2 -16731.687} C_VEL
LIN {X 0,Y 291.583,Z 394.773,A -85,B 0,C 180,E1 -16734.468,E2 -16734.468} C_VEL
LIN {X 0,Y 291.856,Z 394.756,A -85,B 0,C 180,E1 -16738.62,E2 -16738.62} C_VEL
LIN {X 0,Y 291.865,Z 394.729,A -85,B 0,C 180,E1 -16741.38,E2 -16741.38} C_VEL
LIN {X 0,Y 291.683,Z 394.753,A -85,B 0,C 180,E1 -16746.92,E2 -16746.92} C_VEL
LIN {X 0,Y 291.554,Z 394.79,A -85,B 0,C 180,E1 -16749.715,E2 -16749.715} C_VEL
LIN {X 0,Y 291.501,Z 394.796,A -85,B 0,C 180,E1 -16753.951,E2 -16753.951} C_VEL
LIN {X 0,Y 291.414,Z 394.788,A -85,B 0,C 180,E1 -16756.822,E2 -16756.822} C_VEL
LIN {X 0,Y 291.378,Z 394.805,A -85,B 0,C 180,E1 -16759.843,E2 -16759.843} C_VEL
LIN {X 0,Y 291.319,Z 394.814,A -85,B 0,C 180,E1 -16764.213,E2 -16764.213} C_VEL
LIN {X 0,Y 291.315,Z 394.824,A -85,B 0,C 180,E1 -16767.283,E2 -16767.283} C_VEL
LIN {X 0,Y 291.288,Z 394.821,A -85,B 0,C 180,E1 -16770.443,E2 -16770.443} C_VEL
LIN {X 0,Y 291.369,Z 394.87,A -85,B 0,C 180,E1 -16774.364,E2 -16774.364} C_VEL
LIN {X 0,Y 291.56,Z 395.722,A -85,B 0,C 180,E1 -16774.764,E2 -16774.764} C_VEL
LIN {X 0,Y 296.542,Z 406.271,A -85,B 0,C 180,E1 -16778.039,E2 -16778.039} C_VEL
LIN {X 0,Y 301.462,Z 417.706,A -85,B 0,C 180,E1 -16781.27,E2 -16781.27} C_VEL
LIN {X 0,Y 306.298,Z 430.374,A -85,B 0,C 180,E1 -16784.436,E2 -16784.436} C_VEL
LIN {X 0,Y 310.805,Z 444.738,A -85,B 0,C 180,E1 -16787.65,E2 -16787.65} C_VEL
LIN {X 0,Y 314.347,Z 457.97,A -85,B 0,C 180,E1 -16790.335,E2 -16790.335} C_VEL
LIN {X 0,Y 314.713,Z 459.926,A -85,B 0,C 180,E1 -16790.694,E2 -16790.694} C_VEL
LIN {X 0,Y 313.572,Z 470.845,A -85,B 0,C 180,E1 -16792.172,E2 -16792.172} C_VEL
LIN {X 0,Y 318.926,Z 507.717,A -85,B 0,C 180,E1 -16793.942,E2 -16793.942} C_VEL
LIN {X 0,Y 320.07,Z 516.735,A -85,B 0,C 180,E1 -16794.335,E2 -16794.335} C_VEL
LIN {X 0,Y 315.841,Z 628.728,A -85,B 0,C 180,E1 -16796.824,E2 -16796.824} C_VEL
LIN {X 0,Y 314.928,Z 645.999,A -85,B 0,C 180,E1 -16797.287,E2 -16797.287} C_VEL
LIN {X 0,Y 313.564,Z 661.201,A -85,B 0,C 180,E1 -16797.936,E2 -16797.936} C_VEL
LIN {X 0,Y 311.785,Z 675.37,A -85,B 0,C 180,E1 -16798.775,E2 -16798.775} C_VEL
LIN {X 0,Y 309.706,Z 689.306,A -85,B 0,C 180,E1 -16799.866,E2 -16799.866} C_VEL
LIN {X 0,Y 307.124,Z 703.541,A -85,B 0,C 180,E1 -16801.282,E2 -16801.282} C_VEL
LIN {X 0,Y 304.416,Z 716.435,A -85,B 0,C 180,E1 -16802.876,E2 -16802.876} C_VEL
LIN {X 0,Y 302.026,Z 727.262,A -85,B 0,C 180,E1 -16804.504,E2 -16804.504} C_VEL
LIN {X 0,Y 299.515,Z 738.209,A -85,B 0,C 180,E1 -16806.493,E2 -16806.493} C_VEL
LIN {X 0,Y 296.793,Z 748.838,A -85,B 0,C 180,E1 -16808.834,E2 -16808.834} C_VEL
LIN {X 0,Y 294.631,Z 757.679,A -85,B 0,C 180,E1 -16811.217,E2 -16811.217} C_VEL
LIN {X 0,Y 292.815,Z 765.375,A -85,B 0,C 180,E1 -16813.753,E2 -16813.753} C_VEL
LIN {X 0,Y 291.276,Z 772.585,A -85,B 0,C 180,E1 -16816.751,E2 -16816.751} C_VEL
LIN {X 0,Y 290.255,Z 777.777,A -85,B 0,C 180,E1 -16819.539,E2 -16819.539} C_VEL
LIN {X 0,Y 289.797,Z 780.757,A -85,B 0,C 180,E1 -16821.636,E2 -16821.636} C_VEL
LIN {X 0,Y 289.427,Z 783.838,A -85,B 0,C 180,E1 -16824.613,E2 -16824.613} C_VEL
LIN {X 0,Y 289.383,Z 785.453,A -85,B 0,C 180,E1 -16827.218,E2 -16827.218} C_VEL
LIN {X 0,Y 289.351,Z 786.063,A -85,B 0,C 180,E1 -16830.002,E2 -16830.002} C_VEL
LIN {X 0,Y 289.385,Z 785.492,A -85,B 0,C 180,E1 -16832.786,E2 -16832.786} C_VEL
LIN {X 0,Y 289.477,Z 783.781,A -85,B 0,C 180,E1 -16835.575,E2 -16835.575} C_VEL
LIN {X 0,Y 289.805,Z 780.895,A -85,B 0,C 180,E1 -16838.369,E2 -16838.369} C_VEL
LIN {X 0,Y 290.403,Z 776.766,A -85,B 0,C 180,E1 -16841.165,E2 -16841.165} C_VEL
LIN {X 0,Y 291.562,Z 771.297,A -85,B 0,C 180,E1 -16843.95,E2 -16843.95} C_VEL
LIN {X 0,Y 293.03,Z 764.333,A -85,B 0,C 180,E1 -16846.729,E2 -16846.729} C_VEL
LIN {X 0,Y 294.829,Z 756.869,A -85,B 0,C 180,E1 -16849.135,E2 -16849.135} C_VEL
LIN {X 0,Y 297.097,Z 747.876,A -85,B 0,C 180,E1 -16851.512,E2 -16851.512} C_VEL
LIN {X 0,Y 299.56,Z 737.721,A -85,B 0,C 180,E1 -16853.725,E2 -16853.725} C_VEL
LIN {X 0,Y 302.375,Z 725.839,A -85,B 0,C 180,E1 -16855.838,E2 -16855.838} C_VEL
LIN {X 0,Y 305.087,Z 713.576,A -85,B 0,C 180,E1 -16857.622,E2 -16857.622} C_VEL
LIN {X 0,Y 307.854,Z 700.047,A -85,B 0,C 180,E1 -16859.209,E2 -16859.209} C_VEL
LIN {X 0,Y 310.251,Z 686.233,A -85,B 0,C 180,E1 -16860.51,E2 -16860.51} C_VEL
LIN {X 0,Y 312.253,Z 672.12,A -85,B 0,C 180,E1 -16861.556,E2 -16861.556} C_VEL
LIN {X 0,Y 314.003,Z 657.656,A -85,B 0,C 180,E1 -16862.35,E2 -16862.35} C_VEL
LIN {X 0,Y 315.247,Z 643.108,A -85,B 0,C 180,E1 -16862.918,E2 -16862.918} C_VEL
LIN {X 0,Y 316.435,Z 616.888,A -85,B 0,C 180,E1 -16863.539,E2 -16863.539} C_VEL
LIN {X 0,Y 319.861,Z 524.957,A -85,B 0,C 180,E1 -16865.588,E2 -16865.588} C_VEL
LIN {X 0,Y 319.701,Z 521.11,A -85,B 0,C 180,E1 -16865.713,E2 -16865.713} C_VEL
LIN {X 0,Y 318.437,Z 515.607,A -85,B 0,C 180,E1 -16866.026,E2 -16866.026} C_VEL
LIN {X 0,Y 312.37,Z 499.959,A -85,B 0,C 180,E1 -16867.276,E2 -16867.276} C_VEL
LIN {X 0,Y 311.529,Z 496.205,A -85,B 0,C 180,E1 -16867.5,E2 -16867.5} C_VEL
LIN {X 0,Y 307.787,Z 470.485,A -85,B 0,C 180,E1 -16868.823,E2 -16868.823} C_VEL
LIN {X 0,Y 308.593,Z 462.869,A -85,B 0,C 180,E1 -16869.833,E2 -16869.833} C_VEL
LIN {X 0,Y 305.798,Z 450.983,A -85,B 0,C 180,E1 -16872.253,E2 -16872.253} C_VEL
LIN {X 0,Y 301.713,Z 437.552,A -85,B 0,C 180,E1 -16875.265,E2 -16875.265} C_VEL
LIN {X 0,Y 297.08,Z 424.581,A -85,B 0,C 180,E1 -16878.517,E2 -16878.517} C_VEL
LIN {X 0,Y 292.796,Z 414.194,A -85,B 0,C 180,E1 -16881.385,E2 -16881.385} C_VEL
LIN {X 0,Y 287.923,Z 403.352,A -85,B 0,C 180,E1 -16884.713,E2 -16884.713} C_VEL
LIN {X 0,Y 284.389,Z 396.298,A -85,B 0,C 180,E1 -16887.167,E2 -16887.167} C_VEL
LIN {X 0,Y 284.31,Z 395.774,A -85,B 0,C 180,E1 -16887.527,E2 -16887.527} C_VEL
LIN {X 0,Y 284.363,Z 395.879,A -85,B 0,C 180,E1 -16888.578,E2 -16888.578} C_VEL
LIN {X 0,Y 284.785,Z 397.489,A -85,B 0,C 180,E1 -16888.976,E2 -16888.976} C_VEL
LIN {X 0,Y 298.684,Z 434.005,A -85,B 0,C 180,E1 -16891.437,E2 -16891.437} C_VEL
LIN {X 0,Y 293.789,Z 540.526,A -85,B 0,C 180,E1 -16895.194,E2 -16895.194} C_VEL
LIN {X 0,Y 293.239,Z 555.787,A -85,B 0,C 180,E1 -16895.956,E2 -16895.956} C_VEL
LIN {X 0,Y 292.346,Z 571.156,A -85,B 0,C 180,E1 -16897.005,E2 -16897.005} C_VEL
LIN {X 0,Y 291.297,Z 585.158,A -85,B 0,C 180,E1 -16898.226,E2 -16898.226} C_VEL
LIN {X 0,Y 290.183,Z 599.707,A -85,B 0,C 180,E1 -16899.811,E2 -16899.811} C_VEL
LIN {X 0,Y 288.925,Z 612.796,A -85,B 0,C 180,E1 -16901.565,E2 -16901.565} C_VEL
LIN {X 0,Y 287.976,Z 623.772,A -85,B 0,C 180,E1 -16903.336,E2 -16903.336} C_VEL
LIN {X 0,Y 286.871,Z 634.807,A -85,B 0,C 180,E1 -16905.456,E2 -16905.456} C_VEL
LIN {X 0,Y 286.102,Z 644.061,A -85,B 0,C 180,E1 -16907.588,E2 -16907.588} C_VEL
LIN {X 0,Y 285.399,Z 652.977,A -85,B 0,C 180,E1 -16910.074,E2 -16910.074} C_VEL
LIN {X 0,Y 285.04,Z 659.261,A -85,B 0,C 180,E1 -16912.206,E2 -16912.206} C_VEL
LIN {X 0,Y 284.59,Z 664.512,A -85,B 0,C 180,E1 -16914.331,E2 -16914.331} C_VEL
LIN {X 0,Y 284.58,Z 670.024,A -85,B 0,C 180,E1 -16917.169,E2 -16917.169} C_VEL
LIN {X 0,Y 284.764,Z 672.189,A -85,B 0,C 180,E1 -16918.586,E2 -16918.586} C_VEL
LIN {X 0,Y 284.794,Z 673.999,A -85,B 0,C 180,E1 -16920,E2 -16920} C_VEL
LIN {X 0,Y 285.245,Z 675.405,A -85,B 0,C 180,E1 -16921.412,E2 -16921.412} C_VEL
LIN {X 0,Y 286.072,Z 677.184,A -85,B 0,C 180,E1 -16924.226,E2 -16924.226} C_VEL
LIN {X 0,Y 287.149,Z 677.561,A -85,B 0,C 180,E1 -16927.029,E2 -16927.029} C_VEL
LIN {X 0,Y 288.809,Z 676.533,A -85,B 0,C 180,E1 -16929.808,E2 -16929.808} C_VEL
LIN {X 0,Y 290.834,Z 674.123,A -85,B 0,C 180,E1 -16932.561,E2 -16932.561} C_VEL
LIN {X 0,Y 293.492,Z 670.223,A -85,B 0,C 180,E1 -16935.272,E2 -16935.272} C_VEL
LIN {X 0,Y 296.526,Z 664.823,A -85,B 0,C 180,E1 -16937.946,E2 -16937.946} C_VEL
LIN {X 0,Y 300.112,Z 657.69,A -85,B 0,C 180,E1 -16940.565,E2 -16940.565} C_VEL
LIN {X 0,Y 303.61,Z 649.857,A -85,B 0,C 180,E1 -16942.813,E2 -16942.813} C_VEL
LIN {X 0,Y 307.556,Z 640.284,A -85,B 0,C 180,E1 -16945.008,E2 -16945.008} C_VEL
LIN {X 0,Y 311.17,Z 630.531,A -85,B 0,C 180,E1 -16946.854,E2 -16946.854} C_VEL
LIN {X 0,Y 314.713,Z 619.945,A -85,B 0,C 180,E1 -16948.522,E2 -16948.522} C_VEL
LIN {X 0,Y 318.443,Z 607.434,A -85,B 0,C 180,E1 -16950.138,E2 -16950.138} C_VEL
LIN {X 0,Y 322.524,Z 592.151,A -85,B 0,C 180,E1 -16951.697,E2 -16951.697} C_VEL
LIN {X 0,Y 325.604,Z 578.105,A -85,B 0,C 180,E1 -16952.841,E2 -16952.841} C_VEL
LIN {X 0,Y 328.431,Z 562.295,A -85,B 0,C 180,E1 -16953.851,E2 -16953.851} C_VEL
LIN {X 0,Y 331.94,Z 541.662,A -85,B 0,C 180,E1 -16954.866,E2 -16954.866} C_VEL
LIN {X 0,Y 340.091,Z 500.414,A -85,B 0,C 180,E1 -16956.633,E2 -16956.633} C_VEL
LIN {X 0,Y 343.899,Z 482.05,A -85,B 0,C 180,E1 -16957.403,E2 -16957.403} C_VEL
LIN {X 0,Y 342.587,Z 480.07,A -85,B 0,C 180,E1 -16958.779,E2 -16958.779} C_VEL
LIN {X 0,Y 341.464,Z 478.952,A -85,B 0,C 180,E1 -16960.399,E2 -16960.399} C_VEL
LIN {X 0,Y 340.664,Z 479.501,A -85,B 0,C 180,E1 -16962.677,E2 -16962.677} C_VEL
LIN {X 0,Y 340.739,Z 481.305,A -85,B 0,C 180,E1 -16964.398,E2 -16964.398} C_VEL
LIN {X 0,Y 341.274,Z 484.346,A -85,B 0,C 180,E1 -16966.031,E2 -16966.031} C_VEL
LIN {X 0,Y 341.695,Z 486.676,A -85,B 0,C 180,E1 -16966.897,E2 -16966.897} C_VEL
LIN {X 0,Y 341.767,Z 487.799,A -85,B 0,C 180,E1 -16967.164,E2 -16967.164} C_VEL
LIN {X 0,Y 340.149,Z 501.982,A -85,B 0,C 180,E1 -16968.487,E2 -16968.487} C_VEL
LIN {X 0,Y 338.642,Z 514.514,A -85,B 0,C 180,E1 -16969.416,E2 -16969.416} C_VEL
LIN {X 0,Y 337.787,Z 520.551,A -85,B 0,C 180,E1 -16969.766,E2 -16969.766} C_VEL
LIN {X 0,Y 326.431,Z 587.917,A -85,B 0,C 180,E1 -16972.392,E2 -16972.392} C_VEL
LIN {X 0,Y 323.092,Z 606.149,A -85,B 0,C 180,E1 -16973.161,E2 -16973.161} C_VEL
LIN {X 0,Y 318.873,Z 624.268,A -85,B 0,C 180,E1 -16974.164,E2 -16974.164} C_VEL
LIN {X 0,Y 314.503,Z 639.912,A -85,B 0,C 180,E1 -16975.26,E2 -16975.26} C_VEL
LIN {X 0,Y 309.579,Z 655.224,A -85,B 0,C 180,E1 -16976.596,E2 -16976.596} C_VEL
LIN {X 0,Y 306.819,Z 663.61,A -85,B 0,C 180,E1 -16977.479,E2 -16977.479} C_VEL
LIN {X 0,Y 304.911,Z 678.11,A -85,B 0,C 180,E1 -16978.415,E2 -16978.415} C_VEL
LIN {X 0,Y 302.569,Z 692.734,A -85,B 0,C 180,E1 -16979.653,E2 -16979.653} C_VEL
LIN {X 0,Y 299.93,Z 706.226,A -85,B 0,C 180,E1 -16981.098,E2 -16981.098} C_VEL
LIN {X 0,Y 297.051,Z 719.673,A -85,B 0,C 180,E1 -16982.905,E2 -16982.905} C_VEL
LIN {X 0,Y 294.53,Z 729.862,A -85,B 0,C 180,E1 -16984.561,E2 -16984.561} C_VEL
LIN {X 0,Y 292.025,Z 740.255,A -85,B 0,C 180,E1 -16986.601,E2 -16986.601} C_VEL
LIN {X 0,Y 289.353,Z 750.4,A -85,B 0,C 180,E1 -16989.005,E2 -16989.005} C_VEL
LIN {X 0,Y 287.217,Z 758.812,A -85,B 0,C 180,E1 -16991.45,E2 -16991.45} C_VEL
LIN {X 0,Y 285.636,Z 765.113,A -85,B 0,C 180,E1 -16993.654,E2 -16993.654} C_VEL
LIN {X 0,Y 284.287,Z 771.525,A -85,B 0,C 180,E1 -16996.415,E2 -16996.415} C_VEL
LIN {X 0,Y 283.254,Z 776.714,A -85,B 0,C 180,E1 -16999.273,E2 -16999.273} C_VEL
LIN {X 0,Y 282.803,Z 779.699,A -85,B 0,C 180,E1 -17001.423,E2 -17001.423} C_VEL
LIN {X 0,Y 282.436,Z 782.761,A -85,B 0,C 180,E1 -17004.466,E2 -17004.466} C_VEL
LIN {X 0,Y 282.378,Z 784.358,A -85,B 0,C 180,E1 -17007.145,E2 -17007.145} C_VEL
LIN {X 0,Y 282.348,Z 784.949,A -85,B 0,C 180,E1 -17009.998,E2 -17009.998} C_VEL
LIN {X 0,Y 282.382,Z 784.35,A -85,B 0,C 180,E1 -17012.851,E2 -17012.851} C_VEL
LIN {X 0,Y 282.439,Z 782.6,A -85,B 0,C 180,E1 -17015.71,E2 -17015.71} C_VEL
LIN {X 0,Y 282.78,Z 779.673,A -85,B 0,C 180,E1 -17018.574,E2 -17018.574} C_VEL
LIN {X 0,Y 283.421,Z 775.497,A -85,B 0,C 180,E1 -17021.44,E2 -17021.44} C_VEL
LIN {X 0,Y 284.598,Z 769.957,A -85,B 0,C 180,E1 -17024.294,E2 -17024.294} C_VEL
LIN {X 0,Y 286.171,Z 762.903,A -85,B 0,C 180,E1 -17027.137,E2 -17027.137} C_VEL
LIN {X 0,Y 288.055,Z 755.34,A -85,B 0,C 180,E1 -17029.599,E2 -17029.599} C_VEL
LIN {X 0,Y 290.423,Z 746.222,A -85,B 0,C 180,E1 -17032.027,E2 -17032.027} C_VEL
LIN {X 0,Y 292.683,Z 736.925,A -85,B 0,C 180,E1 -17034.09,E2 -17034.09} C_VEL
LIN {X 0,Y 295.449,Z 725.875,A -85,B 0,C 180,E1 -17036.106,E2 -17036.106} C_VEL
LIN {X 0,Y 298.229,Z 713.752,A -85,B 0,C 180,E1 -17037.926,E2 -17037.926} C_VEL
LIN {X 0,Y 301.055,Z 700.402,A -85,B 0,C 180,E1 -17039.545,E2 -17039.545} C_VEL
LIN {X 0,Y 303.618,Z 686.017,A -85,B 0,C 180,E1 -17040.938,E2 -17040.938} C_VEL
LIN {X 0,Y 305.712,Z 671.737,A -85,B 0,C 180,E1 -17042.015,E2 -17042.015} C_VEL
LIN {X 0,Y 307.541,Z 656.335,A -85,B 0,C 180,E1 -17042.868,E2 -17042.868} C_VEL
LIN {X 0,Y 308.764,Z 641.063,A -85,B 0,C 180,E1 -17043.451,E2 -17043.451} C_VEL
LIN {X 0,Y 312.526,Z 547.517,A -85,B 0,C 180,E1 -17045.583,E2 -17045.583} C_VEL
LIN {X 0,Y 313.725,Z 512.361,A -85,B 0,C 180,E1 -17046.398,E2 -17046.398} C_VEL
LIN {X 0,Y 310.216,Z 480.246,A -85,B 0,C 180,E1 -17047.794,E2 -17047.794} C_VEL
LIN {X 0,Y 308.684,Z 466.612,A -85,B 0,C 180,E1 -17048.438,E2 -17048.438} C_VEL
LIN {X 0,Y 308.752,Z 456.603,A -85,B 0,C 180,E1 -17049.292,E2 -17049.292} C_VEL
LIN {X 0,Y 303.161,Z 439.113,A -85,B 0,C 180,E1 -17051.709,E2 -17051.709} C_VEL
LIN {X 0,Y 297.421,Z 422.317,A -85,B 0,C 180,E1 -17054.307,E2 -17054.307} C_VEL
LIN {X 0,Y 294.233,Z 412.964,A -85,B 0,C 180,E1 -17055.885,E2 -17055.885} C_VEL
LIN {X 0,Y 292.238,Z 409.032,A -85,B 0,C 180,E1 -17056.734,E2 -17056.734} C_VEL
LIN {X 0,Y 289.143,Z 404.164,A -85,B 0,C 180,E1 -17057.976,E2 -17057.976} C_VEL
LIN {X 0,Y 286.682,Z 400.172,A -85,B 0,C 180,E1 -17059.022,E2 -17059.022} C_VEL
LIN {X 0,Y 285.047,Z 398.169,A -85,B 0,C 180,E1 -17059.67,E2 -17059.67} C_VEL
LIN {X 0,Y 284.355,Z 396.208,A -85,B 0,C 180,E1 -17060.16,E2 -17060.16} C_VEL
LIN {X 0,Y 284.325,Z 395.727,A -85,B 0,C 180,E1 -17060.469,E2 -17060.469} C_VEL
LIN {X 0,Y 284.324,Z 395.626,A -85,B 0,C 180,E1 -17064.652,E2 -17064.652} C_VEL
LIN {X 0,Y 284.266,Z 395.703,A -85,B 0,C 180,E1 -17068.722,E2 -17068.722} C_VEL
LIN {X 0,Y 284.311,Z 395.697,A -85,B 0,C 180,E1 -17072.854,E2 -17072.854} C_VEL
LIN {X 0,Y 284.293,Z 395.687,A -85,B 0,C 180,E1 -17076.701,E2 -17076.701} C_VEL
LIN {X 0,Y 284.32,Z 395.672,A -85,B 0,C 180,E1 -17079.927,E2 -17079.927} C_VEL
LIN {X 0,Y 284.4,Z 395.662,A -85,B 0,C 180,E1 -17084.516,E2 -17084.516} C_VEL
LIN {X 0,Y 284.464,Z 395.669,A -85,B 0,C 180,E1 -17088.601,E2 -17088.601} C_VEL
LIN {X 0,Y 284.593,Z 395.641,A -85,B 0,C 180,E1 -17091.479,E2 -17091.479} C_VEL
LIN {X 0,Y 284.553,Z 395.65,A -85,B 0,C 180,E1 -17094.33,E2 -17094.33} C_VEL
LIN {X 0,Y 284.823,Z 395.632,A -85,B 0,C 180,E1 -17098.586,E2 -17098.586} C_VEL
LIN {X 0,Y 284.831,Z 395.605,A -85,B 0,C 180,E1 -17101.414,E2 -17101.414} C_VEL
LIN {X 0,Y 284.638,Z 395.631,A -85,B 0,C 180,E1 -17107.092,E2 -17107.092} C_VEL
LIN {X 0,Y 284.5,Z 395.663,A -85,B 0,C 180,E1 -17109.958,E2 -17109.958} C_VEL
LIN {X 0,Y 284.449,Z 395.676,A -85,B 0,C 180,E1 -17114.305,E2 -17114.305} C_VEL
LIN {X 0,Y 284.319,Z 395.692,A -85,B 0,C 180,E1 -17118.744,E2 -17118.744} C_VEL
LIN {X 0,Y 284.296,Z 395.698,A -85,B 0,C 180,E1 -17123.299,E2 -17123.299} C_VEL
LIN {X 0,Y 284.273,Z 395.699,A -85,B 0,C 180,E1 -17127.131,E2 -17127.131} C_VEL
LIN {X 0,Y 284.26,Z 395.692,A -85,B 0,C 180,E1 -17130.085,E2 -17130.085} C_VEL
LIN {X 0,Y 284.296,Z 395.9,A -85,B 0,C 180,E1 -17132.812,E2 -17132.812} C_VEL
LIN {X 0,Y 285.176,Z 398.326,A -85,B 0,C 180,E1 -17133.676,E2 -17133.676} C_VEL
LIN {X 0,Y 286.359,Z 400.099,A -85,B 0,C 180,E1 -17134.366,E2 -17134.366} C_VEL
LIN {X 0,Y 291.524,Z 411.422,A -85,B 0,C 180,E1 -17137.934,E2 -17137.934} C_VEL
LIN {X 0,Y 295.803,Z 421.37,A -85,B 0,C 180,E1 -17140.796,E2 -17140.796} C_VEL
LIN {X 0,Y 300.601,Z 434.168,A -85,B 0,C 180,E1 -17144.071,E2 -17144.071} C_VEL
LIN {X 0,Y 304.703,Z 447.259,A -85,B 0,C 180,E1 -17147.081,E2 -17147.081} C_VEL
LIN {X 0,Y 308.427,Z 461.432,A -85,B 0,C 180,E1 -17149.998,E2 -17149.998} C_VEL
LIN {X 0,Y 308.49,Z 463.709,A -85,B 0,C 180,E1 -17150.368,E2 -17150.368} C_VEL
LIN {X 0,Y 307.779,Z 471.057,A -85,B 0,C 180,E1 -17151.349,E2 -17151.349} C_VEL
LIN {X 0,Y 313.077,Z 507.981,A -85,B 0,C 180,E1 -17153.169,E2 -17153.169} C_VEL
LIN {X 0,Y 314.284,Z 518.031,A -85,B 0,C 180,E1 -17153.613,E2 -17153.613} C_VEL
LIN {X 0,Y 309.936,Z 628.625,A -85,B 0,C 180,E1 -17156.107,E2 -17156.107} C_VEL
LIN {X 0,Y 308.982,Z 645.936,A -85,B 0,C 180,E1 -17156.576,E2 -17156.576} C_VEL
LIN {X 0,Y 307.563,Z 661.157,A -85,B 0,C 180,E1 -17157.233,E2 -17157.233} C_VEL
LIN {X 0,Y 305.72,Z 675.337,A -85,B 0,C 180,E1 -17158.083,E2 -17158.083} C_VEL
LIN {X 0,Y 303.545,Z 689.473,A -85,B 0,C 180,E1 -17159.211,E2 -17159.211} C_VEL
LIN {X 0,Y 300.894,Z 703.518,A -85,B 0,C 180,E1 -17160.629,E2 -17160.629} C_VEL
LIN {X 0,Y 298.09,Z 716.415,A -85,B 0,C 180,E1 -17162.251,E2 -17162.251} C_VEL
LIN {X 0,Y 295.577,Z 727.243,A -85,B 0,C 180,E1 -17163.907,E2 -17163.907} C_VEL
LIN {X 0,Y 292.966,Z 738.193,A -85,B 0,C 180,E1 -17165.935,E2 -17165.935} C_VEL
LIN {X 0,Y 290.149,Z 748.822,A -85,B 0,C 180,E1 -17168.325,E2 -17168.325} C_VEL
LIN {X 0,Y 287.867,Z 757.664,A -85,B 0,C 180,E1 -17170.759,E2 -17170.759} C_VEL
LIN {X 0,Y 285.836,Z 765.791,A -85,B 0,C 180,E1 -17173.519,E2 -17173.519} C_VEL
LIN {X 0,Y 284.31,Z 772.571,A -85,B 0,C 180,E1 -17176.421,E2 -17176.421} C_VEL
LIN {X 0,Y 283.215,Z 777.763,A -85,B 0,C 180,E1 -17179.276,E2 -17179.276} C_VEL
LIN {X 0,Y 282.743,Z 780.744,A -85,B 0,C 180,E1 -17181.425,E2 -17181.425} C_VEL
LIN {X 0,Y 282.348,Z 783.962,A -85,B 0,C 180,E1 -17184.655,E2 -17184.655} C_VEL
LIN {X 0,Y 282.293,Z 785.439,A -85,B 0,C 180,E1 -17187.148,E2 -17187.148} C_VEL
LIN {X 0,Y 282.275,Z 786.05,A -85,B 0,C 180,E1 -17190.002,E2 -17190.002} C_VEL
LIN {X 0,Y 282.295,Z 785.477,A -85,B 0,C 180,E1 -17192.856,E2 -17192.856} C_VEL
LIN {X 0,Y 282.385,Z 783.767,A -85,B 0,C 180,E1 -17195.716,E2 -17195.716} C_VEL
LIN {X 0,Y 282.748,Z 780.88,A -85,B 0,C 180,E1 -17198.579,E2 -17198.579} C_VEL
LIN {X 0,Y 283.379,Z 776.75,A -85,B 0,C 180,E1 -17201.446,E2 -17201.446} C_VEL
LIN {X 0,Y 284.608,Z 771.28,A -85,B 0,C 180,E1 -17204.298,E2 -17204.298} C_VEL
LIN {X 0,Y 286.184,Z 764.315,A -85,B 0,C 180,E1 -17207.141,E2 -17207.141} C_VEL
LIN {X 0,Y 288.074,Z 756.85,A -85,B 0,C 180,E1 -17209.602,E2 -17209.602} C_VEL
LIN {X 0,Y 290.471,Z 747.855,A -85,B 0,C 180,E1 -17212.028,E2 -17212.028} C_VEL
LIN {X 0,Y 293.151,Z 737.34,A -85,B 0,C 180,E1 -17214.354,E2 -17214.354} C_VEL
LIN {X 0,Y 295.967,Z 725.814,A -85,B 0,C 180,E1 -17216.44,E2 -17216.44} C_VEL
LIN {X 0,Y 298.808,Z 713.546,A -85,B 0,C 180,E1 -17218.253,E2 -17218.253} C_VEL
LIN {X 0,Y 301.667,Z 700.013,A -85,B 0,C 180,E1 -17219.868,E2 -17219.868} C_VEL
LIN {X 0,Y 303.975,Z 687.338,A -85,B 0,C 180,E1 -17221.094,E2 -17221.094} C_VEL
LIN {X 0,Y 306.073,Z 673.307,A -85,B 0,C 180,E1 -17222.172,E2 -17222.172} C_VEL
LIN {X 0,Y 307.949,Z 658.438,A -85,B 0,C 180,E1 -17223.018,E2 -17223.018} C_VEL
LIN {X 0,Y 309.323,Z 642.998,A -85,B 0,C 180,E1 -17223.631,E2 -17223.631} C_VEL
LIN {X 0,Y 310.715,Z 611.38,A -85,B 0,C 180,E1 -17224.388,E2 -17224.388} C_VEL
LIN {X 0,Y 314.371,Z 517.473,A -85,B 0,C 180,E1 -17226.511,E2 -17226.511} C_VEL
LIN {X 0,Y 311.529,Z 496.205,A -85,B 0,C 180,E1 -17227.5,E2 -17227.5} C_VEL
LIN {X 0,Y 310.412,Z 492.635,A -85,B 0,C 180,E1 -17227.76,E2 -17227.76} C_VEL
LIN {X 0,Y 304.264,Z 482.461,A -85,B 0,C 180,E1 -17228.959,E2 -17228.959} C_VEL
LIN {X 0,Y 303.275,Z 478.863,A -85,B 0,C 180,E1 -17229.217,E2 -17229.217} C_VEL
LIN {X 0,Y 302.014,Z 471.001,A -85,B 0,C 180,E1 -17229.653,E2 -17229.653} C_VEL
LIN {X 0,Y 302.59,Z 465.44,A -85,B 0,C 180,E1 -17230.37,E2 -17230.37} C_VEL
LIN {X 0,Y 300.154,Z 455.216,A -85,B 0,C 180,E1 -17232.477,E2 -17232.477} C_VEL
LIN {X 0,Y 296.387,Z 442.499,A -85,B 0,C 180,E1 -17235.349,E2 -17235.349} C_VEL
LIN {X 0,Y 292.033,Z 429.864,A -85,B 0,C 180,E1 -17238.561,E2 -17238.561} C_VEL
LIN {X 0,Y 288.121,Z 419.978,A -85,B 0,C 180,E1 -17241.314,E2 -17241.314} C_VEL
LIN {X 0,Y 283.148,Z 408.852,A -85,B 0,C 180,E1 -17244.754,E2 -17244.754} C_VEL
LIN {X 0,Y 278.561,Z 399.818,A -85,B 0,C 180,E1 -17248.006,E2 -17248.006} C_VEL
LIN {X 0,Y 278.305,Z 399.427,A -85,B 0,C 180,E1 -17248.281,E2 -17248.281} C_VEL
LIN {X 0,Y 278.39,Z 399.804,A -85,B 0,C 180,E1 -17248.488,E2 -17248.488} C_VEL
LIN {X 0,Y 279.251,Z 402.206,A -85,B 0,C 180,E1 -17248.752,E2 -17248.752} C_VEL
LIN {X 0,Y 291.917,Z 435.627,A -85,B 0,C 180,E1 -17251.046,E2 -17251.046} C_VEL
LIN {X 0,Y 286.893,Z 540.566,A -85,B 0,C 180,E1 -17254.863,E2 -17254.863} C_VEL
LIN {X 0,Y 286.332,Z 555.747,A -85,B 0,C 180,E1 -17255.628,E2 -17255.628} C_VEL
LIN {X 0,Y 285.429,Z 571.378,A -85,B 0,C 180,E1 -17256.703,E2 -17256.703} C_VEL
LIN {X 0,Y 284.302,Z 586.422,A -85,B 0,C 180,E1 -17258.044,E2 -17258.044} C_VEL
LIN {X 0,Y 283.132,Z 600.922,A -85,B 0,C 180,E1 -17259.665,E2 -17259.665} C_VEL
LIN {X 0,Y 281.806,Z 614.596,A -85,B 0,C 180,E1 -17261.558,E2 -17261.558} C_VEL
LIN {X 0,Y 280.883,Z 624.909,A -85,B 0,C 180,E1 -17263.277,E2 -17263.277} C_VEL
LIN {X 0,Y 279.763,Z 635.898,A -85,B 0,C 180,E1 -17265.451,E2 -17265.451} C_VEL
LIN {X 0,Y 278.995,Z 645.125,A -85,B 0,C 180,E1 -17267.636,E2 -17267.636} C_VEL
LIN {X 0,Y 278.344,Z 653.418,A -85,B 0,C 180,E1 -17269.981,E2 -17269.981} C_VEL
LIN {X 0,Y 277.98,Z 659.424,A -85,B 0,C 180,E1 -17272.007,E2 -17272.007} C_VEL
LIN {X 0,Y 277.55,Z 664.9,A -85,B 0,C 180,E1 -17274.187,E2 -17274.187} C_VEL
LIN {X 0,Y 277.512,Z 670.611,A -85,B 0,C 180,E1 -17277.097,E2 -17277.097} C_VEL
LIN {X 0,Y 277.712,Z 672.862,A -85,B 0,C 180,E1 -17278.55,E2 -17278.55} C_VEL
LIN {X 0,Y 277.742,Z 674.767,A -85,B 0,C 180,E1 -17280,E2 -17280} C_VEL
LIN {X 0,Y 278.211,Z 676.282,A -85,B 0,C 180,E1 -17281.447,E2 -17281.447} C_VEL
LIN {X 0,Y 279.091,Z 678.288,A -85,B 0,C 180,E1 -17284.332,E2 -17284.332} C_VEL
LIN {X 0,Y 280.251,Z 678.918,A -85,B 0,C 180,E1 -17287.203,E2 -17287.203} C_VEL
LIN {X 0,Y 282.002,Z 678.131,A -85,B 0,C 180,E1 -17290.047,E2 -17290.047} C_VEL
LIN {X 0,Y 284.17,Z 675.956,A -85,B 0,C 180,E1 -17292.861,E2 -17292.861} C_VEL
LIN {X 0,Y 286.977,Z 672.313,A -85,B 0,C 180,E1 -17295.628,E2 -17295.628} C_VEL
LIN {X 0,Y 290.163,Z 667.19,A -85,B 0,C 180,E1 -17298.353,E2 -17298.353} C_VEL
LIN {X 0,Y 292.974,Z 662.281,A -85,B 0,C 180,E1 -17300.355,E2 -17300.355} C_VEL
LIN {X 0,Y 297.081,Z 654.129,A -85,B 0,C 180,E1 -17302.975,E2 -17302.975} C_VEL
LIN {X 0,Y 300.552,Z 646.67,A -85,B 0,C 180,E1 -17304.892,E2 -17304.892} C_VEL
LIN {X 0,Y 304.942,Z 636.308,A -85,B 0,C 180,E1 -17307.076,E2 -17307.076} C_VEL
LIN {X 0,Y 308.954,Z 625.665,A -85,B 0,C 180,E1 -17308.907,E2 -17308.907} C_VEL
LIN {X 0,Y 313.412,Z 612.506,A -85,B 0,C 180,E1 -17310.746,E2 -17310.746} C_VEL
LIN {X 0,Y 317.372,Z 599.425,A -85,B 0,C 180,E1 -17312.208,E2 -17312.208} C_VEL
LIN {X 0,Y 321.127,Z 584.629,A -85,B 0,C 180,E1 -17313.546,E2 -17313.546} C_VEL
LIN {X 0,Y 324.54,Z 568.62,A -85,B 0,C 180,E1 -17314.656,E2 -17314.656} C_VEL
LIN {X 0,Y 327.803,Z 550.222,A -85,B 0,C 180,E1 -17315.654,E2 -17315.654} C_VEL
LIN {X 0,Y 337.917,Z 501.829,A -85,B 0,C 180,E1 -17317.752,E2 -17317.752} C_VEL
LIN {X 0,Y 341.039,Z 487.57,A -85,B 0,C 180,E1 -17318.358,E2 -17318.358} C_VEL
LIN {X 0,Y 340.243,Z 486.47,A -85,B 0,C 180,E1 -17319.371,E2 -17319.371} C_VEL
LIN {X 0,Y 339.804,Z 485.963,A -85,B 0,C 180,E1 -17320.069,E2 -17320.069} C_VEL
LIN {X 0,Y 338.915,Z 486.114,A -85,B 0,C 180,E1 -17322.202,E2 -17322.202} C_VEL
LIN {X 0,Y 338.822,Z 487.838,A -85,B 0,C 180,E1 -17324.072,E2 -17324.072} C_VEL
LIN {X 0,Y 339.239,Z 491.006,A -85,B 0,C 180,E1 -17325.775,E2 -17325.775} C_VEL
LIN {X 0,Y 339.413,Z 492.535,A -85,B 0,C 180,E1 -17326.324,E2 -17326.324} C_VEL
LIN {X 0,Y 337.505,Z 506.101,A -85,B 0,C 180,E1 -17327.574,E2 -17327.574} C_VEL
LIN {X 0,Y 335.727,Z 518.356,A -85,B 0,C 180,E1 -17328.476,E2 -17328.476} C_VEL
LIN {X 0,Y 334.849,Z 523.385,A -85,B 0,C 180,E1 -17328.729,E2 -17328.729} C_VEL
LIN {X 0,Y 323.345,Z 586.748,A -85,B 0,C 180,E1 -17331.224,E2 -17331.224} C_VEL
LIN {X 0,Y 319.714,Z 605.004,A -85,B 0,C 180,E1 -17332.01,E2 -17332.01} C_VEL
LIN {X 0,Y 315.573,Z 621.661,A -85,B 0,C 180,E1 -17332.935,E2 -17332.935} C_VEL
LIN {X 0,Y 310.461,Z 638.91,A -85,B 0,C 180,E1 -17334.143,E2 -17334.143} C_VEL
LIN {X 0,Y 305.33,Z 653.917,A -85,B 0,C 180,E1 -17335.47,E2 -17335.47} C_VEL
LIN {X 0,Y 300.362,Z 667.727,A -85,B 0,C 180,E1 -17336.991,E2 -17336.991} C_VEL
LIN {X 0,Y 298.165,Z 682.619,A -85,B 0,C 180,E1 -17338.054,E2 -17338.054} C_VEL
LIN {X 0,Y 295.874,Z 695.963,A -85,B 0,C 180,E1 -17339.288,E2 -17339.288} C_VEL
LIN {X 0,Y 293.164,Z 708.864,A -85,B 0,C 180,E1 -17340.759,E2 -17340.759} C_VEL
LIN {X 0,Y 290.451,Z 720.761,A -85,B 0,C 180,E1 -17342.432,E2 -17342.432} C_VEL
LIN {X 0,Y 287.612,Z 731.768,A -85,B 0,C 180,E1 -17344.294,E2 -17344.294} C_VEL
LIN {X 0,Y 285.041,Z 741.993,A -85,B 0,C 180,E1 -17346.405,E2 -17346.405} C_VEL
LIN {X 0,Y 282.367,Z 751.754,A -85,B 0,C 180,E1 -17348.843,E2 -17348.843} C_VEL
LIN {X 0,Y 280.15,Z 759.94,A -85,B 0,C 180,E1 -17351.344,E2 -17351.344} C_VEL
LIN {X 0,Y 278.427,Z 766.701,A -85,B 0,C 180,E1 -17353.877,E2 -17353.877} C_VEL
LIN {X 0,Y 277.008,Z 772.957,A -85,B 0,C 180,E1 -17356.799,E2 -17356.799} C_VEL
LIN {X 0,Y 276.065,Z 777.79,A -85,B 0,C 180,E1 -17359.733,E2 -17359.733} C_VEL
LIN {X 0,Y 275.519,Z 781.326,A -85,B 0,C 180,E1 -17362.67,E2 -17362.67} C_VEL
LIN {X 0,Y 275.288,Z 783.648,A -85,B 0,C 180,E1 -17365.605,E2 -17365.605} C_VEL
LIN {X 0,Y 275.277,Z 784.812,A -85,B 0,C 180,E1 -17368.535,E2 -17368.535} C_VEL
LIN {X 0,Y 275.279,Z 784.809,A -85,B 0,C 180,E1 -17371.461,E2 -17371.461} C_VEL
LIN {X 0,Y 275.283,Z 783.633,A -85,B 0,C 180,E1 -17374.39,E2 -17374.39} C_VEL
LIN {X 0,Y 275.51,Z 781.301,A -85,B 0,C 180,E1 -17377.325,E2 -17377.325} C_VEL
LIN {X 0,Y 276.054,Z 777.761,A -85,B 0,C 180,E1 -17380.263,E2 -17380.263} C_VEL
LIN {X 0,Y 277,Z 772.92,A -85,B 0,C 180,E1 -17383.197,E2 -17383.197} C_VEL
LIN {X 0,Y 278.414,Z 766.645,A -85,B 0,C 180,E1 -17386.119,E2 -17386.119} C_VEL
LIN {X 0,Y 280.418,Z 758.759,A -85,B 0,C 180,E1 -17389.012,E2 -17389.012} C_VEL
LIN {X 0,Y 282.651,Z 750.339,A -85,B 0,C 180,E1 -17391.513,E2 -17391.513} C_VEL
LIN {X 0,Y 285.323,Z 740.576,A -85,B 0,C 180,E1 -17393.882,E2 -17393.882} C_VEL
LIN {X 0,Y 287.122,Z 733.428,A -85,B 0,C 180,E1 -17395.36,E2 -17395.36} C_VEL
LIN {X 0,Y 290.106,Z 721.698,A -85,B 0,C 180,E1 -17397.403,E2 -17397.403} C_VEL
LIN {X 0,Y 292.835,Z 709.99,A -85,B 0,C 180,E1 -17399.075,E2 -17399.075} C_VEL
LIN {X 0,Y 295.451,Z 697.325,A -85,B 0,C 180,E1 -17400.558,E2 -17400.558} C_VEL
LIN {X 0,Y 298.014,Z 682.95,A -85,B 0,C 180,E1 -17401.899,E2 -17401.899} C_VEL
LIN {X 0,Y 300.2,Z 667.941,A -85,B 0,C 180,E1 -17402.974,E2 -17402.974} C_VEL
LIN {X 0,Y 301.943,Z 652.803,A -85,B 0,C 180,E1 -17403.757,E2 -17403.757} C_VEL
LIN {X 0,Y 303.093,Z 638.243,A -85,B 0,C 180,E1 -17404.262,E2 -17404.262} C_VEL
LIN {X 0,Y 307.017,Z 542.004,A -85,B 0,C 180,E1 -17406.482,E2 -17406.482} C_VEL
LIN {X 0,Y 308.023,Z 513.327,A -85,B 0,C 180,E1 -17407.159,E2 -17407.159} C_VEL
LIN {X 0,Y 304.326,Z 478.314,A -85,B 0,C 180,E1 -17408.72,E2 -17408.72} C_VEL
LIN {X 0,Y 303.016,Z 466.442,A -85,B 0,C 180,E1 -17409.315,E2 -17409.315} C_VEL
LIN {X 0,Y 303.117,Z 459.489,A -85,B 0,C 180,E1 -17409.915,E2 -17409.915} C_VEL
LIN {X 0,Y 297.528,Z 441.472,A -85,B 0,C 180,E1 -17412.513,E2 -17412.513} C_VEL
LIN {X 0,Y 292.486,Z 426.304,A -85,B 0,C 180,E1 -17414.929,E2 -17414.929} C_VEL
LIN {X 0,Y 289.819,Z 417.978,A -85,B 0,C 180,E1 -17416.378,E2 -17416.378} C_VEL
LIN {X 0,Y 287.686,Z 413.739,A -85,B 0,C 180,E1 -17417.319,E2 -17417.319} C_VEL
LIN {X 0,Y 282.992,Z 406.103,A -85,B 0,C 180,E1 -17419.314,E2 -17419.314} C_VEL
LIN {X 0,Y 280.783,Z 403.062,A -85,B 0,C 180,E1 -17420.242,E2 -17420.242} C_VEL
LIN {X 0,Y 280.316,Z 401.895,A -85,B 0,C 180,E1 -17420.505,E2 -17420.505} C_VEL
LIN {X 0,Y 277.758,Z 398.425,A -85,B 0,C 180,E1 -17421.659,E2 -17421.659} C_VEL
LIN {X 0,Y 277.31,Z 396.852,A -85,B 0,C 180,E1 -17422.155,E2 -17422.155} C_VEL
LIN {X 0,Y 277.245,Z 396.559,A -85,B 0,C 180,E1 -17422.527,E2 -17422.527} C_VEL
LIN {X 0,Y 277.233,Z 396.517,A -85,B 0,C 180,E1 -17426.103,E2 -17426.103} C_VEL
LIN {X 0,Y 277.215,Z 396.569,A -85,B 0,C 180,E1 -17429.533,E2 -17429.533} C_VEL
LIN {X 0,Y 277.273,Z 396.573,A -85,B 0,C 180,E1 -17432.855,E2 -17432.855} C_VEL
LIN {X 0,Y 277.241,Z 396.558,A -85,B 0,C 180,E1 -17436.072,E2 -17436.072} C_VEL
LIN {X 0,Y 277.264,Z 396.553,A -85,B 0,C 180,E1 -17440.761,E2 -17440.761} C_VEL
LIN {X 0,Y 277.356,Z 396.537,A -85,B 0,C 180,E1 -17445.322,E2 -17445.322} C_VEL
LIN {X 0,Y 277.442,Z 396.527,A -85,B 0,C 180,E1 -17449.786,E2 -17449.786} C_VEL
LIN {X 0,Y 277.584,Z 396.53,A -85,B 0,C 180,E1 -17452.727,E2 -17452.727} C_VEL
LIN {X 0,Y 277.79,Z 396.509,A -85,B 0,C 180,E1 -17458.55,E2 -17458.55} C_VEL
LIN {X 0,Y 277.797,Z 396.481,A -85,B 0,C 180,E1 -17461.45,E2 -17461.45} C_VEL
LIN {X 0,Y 277.596,Z 396.508,A -85,B 0,C 180,E1 -17467.273,E2 -17467.273} C_VEL
LIN {X 0,Y 277.441,Z 396.538,A -85,B 0,C 180,E1 -17470.214,E2 -17470.214} C_VEL
LIN {X 0,Y 277.395,Z 396.551,A -85,B 0,C 180,E1 -17474.676,E2 -17474.676} C_VEL
LIN {X 0,Y 277.271,Z 396.57,A -85,B 0,C 180,E1 -17479.239,E2 -17479.239} C_VEL
LIN {X 0,Y 277.247,Z 396.57,A -85,B 0,C 180,E1 -17483.928,E2 -17483.928} C_VEL
LIN {X 0,Y 277.222,Z 396.58,A -85,B 0,C 180,E1 -17487.47,E2 -17487.47} C_VEL
LIN {X 0,Y 277.24,Z 396.781,A -85,B 0,C 180,E1 -17490.992,E2 -17490.992} C_VEL
LIN {X 0,Y 278.311,Z 399.458,A -85,B 0,C 180,E1 -17492.026,E2 -17492.026} C_VEL
LIN {X 0,Y 279.547,Z 401.632,A -85,B 0,C 180,E1 -17492.864,E2 -17492.864} C_VEL
LIN {X 0,Y 282.935,Z 408.485,A -85,B 0,C 180,E1 -17495.277,E2 -17495.277} C_VEL
LIN {X 0,Y 287.646,Z 419.058,A -85,B 0,C 180,E1 -17498.574,E2 -17498.574} C_VEL
LIN {X 0,Y 291.208,Z 427.799,A -85,B 0,C 180,E1 -17501.051,E2 -17501.051} C_VEL
LIN {X 0,Y 295.472,Z 439.588,A -85,B 0,C 180,E1 -17504.085,E2 -17504.085} C_VEL
LIN {X 0,Y 299.682,Z 453.733,A -85,B 0,C 180,E1 -17507.33,E2 -17507.33} C_VEL
LIN {X 0,Y 302.509,Z 464.732,A -85,B 0,C 180,E1 -17509.61,E2 -17509.61} C_VEL
LIN {X 0,Y 301.954,Z 470.786,A -85,B 0,C 180,E1 -17510.448,E2 -17510.448} C_VEL
LIN {X 0,Y 306.771,Z 504.485,A -85,B 0,C 180,E1 -17512.184,E2 -17512.184} C_VEL
LIN {X 0,Y 308.543,Z 519.411,A -85,B 0,C 180,E1 -17512.867,E2 -17512.867} C_VEL
LIN {X 0,Y 303.987,Z 630.305,A -85,B 0,C 180,E1 -17515.401,E2 -17515.401} C_VEL
LIN {X 0,Y 303.014,Z 646.94,A -85,B 0,C 180,E1 -17515.878,E2 -17515.878} C_VEL
LIN {X 0,Y 301.463,Z 662.572,A -85,B 0,C 180,E1 -17516.583,E2 -17516.583} C_VEL
LIN {X 0,Y 299.469,Z 676.908,A -85,B 0,C 180,E1 -17517.482,E2 -17517.482} C_VEL
LIN {X 0,Y 297.165,Z 690.967,A -85,B 0,C 180,E1 -17518.65,E2 -17518.65} C_VEL
LIN {X 0,Y 294.414,Z 704.892,A -85,B 0,C 180,E1 -17520.115,E2 -17520.115} C_VEL
LIN {X 0,Y 291.517,Z 717.548,A -85,B 0,C 180,E1 -17521.765,E2 -17521.765} C_VEL
LIN {X 0,Y 288.701,Z 729.145,A -85,B 0,C 180,E1 -17523.626,E2 -17523.626} C_VEL
LIN {X 0,Y 286.047,Z 739.781,A -85,B 0,C 180,E1 -17525.701,E2 -17525.701} C_VEL
LIN {X 0,Y 283.103,Z 750.142,A -85,B 0,C 180,E1 -17528.141,E2 -17528.141} C_VEL
LIN {X 0,Y 280.804,Z 758.752,A -85,B 0,C 180,E1 -17530.635,E2 -17530.635} C_VEL
LIN {X 0,Y 278.863,Z 766.201,A -85,B 0,C 180,E1 -17533.274,E2 -17533.274} C_VEL
LIN {X 0,Y 277.358,Z 772.557,A -85,B 0,C 180,E1 -17536.073,E2 -17536.073} C_VEL
LIN {X 0,Y 276.191,Z 777.749,A -85,B 0,C 180,E1 -17539,E2 -17539} C_VEL
LIN {X 0,Y 275.683,Z 780.73,A -85,B 0,C 180,E1 -17541.204,E2 -17541.204} C_VEL
LIN {X 0,Y 275.289,Z 783.663,A -85,B 0,C 180,E1 -17544.141,E2 -17544.141} C_VEL
LIN {X 0,Y 275.204,Z 785.425,A -85,B 0,C 180,E1 -17547.075,E2 -17547.075} C_VEL
LIN {X 0,Y 275.2,Z 786.036,A -85,B 0,C 180,E1 -17550.002,E2 -17550.002} C_VEL
LIN {X 0,Y 275.207,Z 785.463,A -85,B 0,C 180,E1 -17552.93,E2 -17552.93} C_VEL
LIN {X 0,Y 275.298,Z 783.752,A -85,B 0,C 180,E1 -17555.863,E2 -17555.863} C_VEL
LIN {X 0,Y 275.686,Z 780.865,A -85,B 0,C 180,E1 -17558.8,E2 -17558.8} C_VEL
LIN {X 0,Y 276.369,Z 776.734,A -85,B 0,C 180,E1 -17561.74,E2 -17561.74} C_VEL
LIN {X 0,Y 277.655,Z 771.263,A -85,B 0,C 180,E1 -17564.664,E2 -17564.664} C_VEL
LIN {X 0,Y 279.338,Z 764.297,A -85,B 0,C 180,E1 -17567.575,E2 -17567.575} C_VEL
LIN {X 0,Y 281.347,Z 756.831,A -85,B 0,C 180,E1 -17570.091,E2 -17570.091} C_VEL
LIN {X 0,Y 283.869,Z 747.834,A -85,B 0,C 180,E1 -17572.568,E2 -17572.568} C_VEL
LIN {X 0,Y 286.709,Z 737.139,A -85,B 0,C 180,E1 -17574.977,E2 -17574.977} C_VEL
LIN {X 0,Y 289.599,Z 725.788,A -85,B 0,C 180,E1 -17577.069,E2 -17577.069} C_VEL
LIN {X 0,Y 292.556,Z 713.517,A -85,B 0,C 180,E1 -17578.913,E2 -17578.913} C_VEL
LIN {X 0,Y 295.223,Z 701.507,A -85,B 0,C 180,E1 -17580.391,E2 -17580.391} C_VEL
LIN {X 0,Y 297.898,Z 687.324,A -85,B 0,C 180,E1 -17581.799,E2 -17581.799} C_VEL
LIN {X 0,Y 300.075,Z 673.256,A -85,B 0,C 180,E1 -17582.895,E2 -17582.895} C_VEL
LIN {X 0,Y 302.036,Z 658.369,A -85,B 0,C 180,E1 -17583.75,E2 -17583.75} C_VEL
LIN {X 0,Y 303.449,Z 642.885,A -85,B 0,C 180,E1 -17584.372,E2 -17584.372} C_VEL
LIN {X 0,Y 304.888,Z 611.229,A -85,B 0,C 180,E1 -17585.141,E2 -17585.141} C_VEL
LIN {X 0,Y 308.666,Z 518.628,A -85,B 0,C 180,E1 -17587.262,E2 -17587.262} C_VEL
LIN {X 0,Y 304.371,Z 486.592,A -85,B 0,C 180,E1 -17588.82,E2 -17588.82} C_VEL
LIN {X 0,Y 303.275,Z 478.863,A -85,B 0,C 180,E1 -17589.217,E2 -17589.217} C_VEL
LIN {X 0,Y 302.584,Z 475.266,A -85,B 0,C 180,E1 -17589.473,E2 -17589.473} C_VEL
LIN {X 0,Y 300.89,Z 470.568,A -85,B 0,C 180,E1 -17590.07,E2 -17590.07} C_VEL
LIN {X 0,Y 298.83,Z 466.626,A -85,B 0,C 180,E1 -17590.832,E2 -17590.832} C_VEL
LIN {X 0,Y 296.001,Z 461.866,A -85,B 0,C 180,E1 -17592.026,E2 -17592.026} C_VEL
LIN {X 0,Y 293.87,Z 456.969,A -85,B 0,C 180,E1 -17593.26,E2 -17593.26} C_VEL
LIN {X 0,Y 290.489,Z 445.517,A -85,B 0,C 180,E1 -17595.928,E2 -17595.928} C_VEL
LIN {X 0,Y 286.465,Z 433.759,A -85,B 0,C 180,E1 -17598.984,E2 -17598.984} C_VEL
LIN {X 0,Y 282.371,Z 423.342,A -85,B 0,C 180,E1 -17601.975,E2 -17601.975} C_VEL
LIN {X 0,Y 277.465,Z 412.181,A -85,B 0,C 180,E1 -17605.549,E2 -17605.549} C_VEL
LIN {X 0,Y 274.623,Z 406.497,A -85,B 0,C 180,E1 -17607.623,E2 -17607.623} C_VEL
LIN {X 0,Y 273.867,Z 405.616,A -85,B 0,C 180,E1 -17608.11,E2 -17608.11} C_VEL
LIN {X 0,Y 273.65,Z 406.424,A -85,B 0,C 180,E1 -17608.414,E2 -17608.414} C_VEL
LIN {X 0,Y 275.073,Z 410.392,A -85,B 0,C 180,E1 -17608.776,E2 -17608.776} C_VEL
LIN {X 0,Y 285.139,Z 437.112,A -85,B 0,C 180,E1 -17610.641,E2 -17610.641} C_VEL
LIN {X 0,Y 280.011,Z 541.077,A -85,B 0,C 180,E1 -17614.537,E2 -17614.537} C_VEL
LIN {X 0,Y 279.388,Z 557.303,A -85,B 0,C 180,E1 -17615.378,E2 -17615.378} C_VEL
LIN {X 0,Y 278.455,Z 572.629,A -85,B 0,C 180,E1 -17616.478,E2 -17616.478} C_VEL
LIN {X 0,Y 277.294,Z 587.522,A -85,B 0,C 180,E1 -17617.851,E2 -17617.851} C_VEL
LIN {X 0,Y 276.088,Z 601.93,A -85,B 0,C 180,E1 -17619.512,E2 -17619.512} C_VEL
LIN {X 0,Y 274.824,Z 614.462,A -85,B 0,C 180,E1 -17621.279,E2 -17621.279} C_VEL
LIN {X 0,Y 273.78,Z 625.889,A -85,B 0,C 180,E1 -17623.214,E2 -17623.214} C_VEL
LIN {X 0,Y 272.674,Z 636.922,A -85,B 0,C 180,E1 -17625.445,E2 -17625.445} C_VEL
LIN {X 0,Y 271.887,Z 646.196,A -85,B 0,C 180,E1 -17627.687,E2 -17627.687} C_VEL
LIN {X 0,Y 271.204,Z 655.224,A -85,B 0,C 180,E1 -17630.31,E2 -17630.31} C_VEL
LIN {X 0,Y 270.787,Z 661.533,A -85,B 0,C 180,E1 -17632.544,E2 -17632.544} C_VEL
LIN {X 0,Y 270.407,Z 668.384,A -85,B 0,C 180,E1 -17635.528,E2 -17635.528} C_VEL
LIN {X 0,Y 270.66,Z 673.518,A -85,B 0,C 180,E1 -17638.512,E2 -17638.512} C_VEL
LIN {X 0,Y 270.691,Z 675.535,A -85,B 0,C 180,E1 -17640,E2 -17640} C_VEL
LIN {X 0,Y 271.176,Z 677.157,A -85,B 0,C 180,E1 -17641.485,E2 -17641.485} C_VEL
LIN {X 0,Y 272.108,Z 679.362,A -85,B 0,C 180,E1 -17644.444,E2 -17644.444} C_VEL
LIN {X 0,Y 273.349,Z 680.211,A -85,B 0,C 180,E1 -17647.386,E2 -17647.386} C_VEL
LIN {X 0,Y 275.188,Z 679.661,A -85,B 0,C 180,E1 -17650.298,E2 -17650.298} C_VEL
LIN {X 0,Y 277.494,Z 677.768,A -85,B 0,C 180,E1 -17653.176,E2 -17653.176} C_VEL
LIN {X 0,Y 280.448,Z 674.422,A -85,B 0,C 180,E1 -17656.001,E2 -17656.001} C_VEL
LIN {X 0,Y 283.826,Z 669.62,A -85,B 0,C 180,E1 -17658.778,E2 -17658.778} C_VEL
LIN {X 0,Y 287.813,Z 663.156,A -85,B 0,C 180,E1 -17661.486,E2 -17661.486} C_VEL
LIN {X 0,Y 292.3,Z 655.002,A -85,B 0,C 180,E1 -17664.126,E2 -17664.126} C_VEL
LIN {X 0,Y 296.72,Z 646.155,A -85,B 0,C 180,E1 -17666.366,E2 -17666.366} C_VEL
LIN {X 0,Y 301.456,Z 635.502,A -85,B 0,C 180,E1 -17668.55,E2 -17668.55} C_VEL
LIN {X 0,Y 305.831,Z 624.621,A -85,B 0,C 180,E1 -17670.368,E2 -17670.368} C_VEL
LIN {X 0,Y 310.11,Z 612.817,A -85,B 0,C 180,E1 -17671.988,E2 -17671.988} C_VEL
LIN {X 0,Y 314.772,Z 598.259,A -85,B 0,C 180,E1 -17673.572,E2 -17673.572} C_VEL
LIN {X 0,Y 318.79,Z 583.409,A -85,B 0,C 180,E1 -17674.877,E2 -17674.877} C_VEL
LIN {X 0,Y 322.464,Z 566.569,A -85,B 0,C 180,E1 -17675.999,E2 -17675.999} C_VEL
LIN {X 0,Y 326.412,Z 546.623,A -85,B 0,C 180,E1 -17677.027,E2 -17677.027} C_VEL
LIN {X 0,Y 336.51,Z 501.589,A -85,B 0,C 180,E1 -17678.953,E2 -17678.953} C_VEL
LIN {X 0,Y 338.411,Z 493.388,A -85,B 0,C 180,E1 -17679.326,E2 -17679.326} C_VEL
LIN {X 0,Y 337.902,Z 492.815,A -85,B 0,C 180,E1 -17680.148,E2 -17680.148} C_VEL
LIN {X 0,Y 337.082,Z 492.983,A -85,B 0,C 180,E1 -17682.18,E2 -17682.18} C_VEL
LIN {X 0,Y 336.938,Z 494.619,A -85,B 0,C 180,E1 -17683.874,E2 -17683.874} C_VEL
LIN {X 0,Y 337.205,Z 497.646,A -85,B 0,C 180,E1 -17685.494,E2 -17685.494} C_VEL
LIN {X 0,Y 335.012,Z 510.688,A -85,B 0,C 180,E1 -17686.678,E2 -17686.678} C_VEL
LIN {X 0,Y 333.077,Z 522.135,A -85,B 0,C 180,E1 -17687.498,E2 -17687.498} C_VEL
LIN {X 0,Y 317.893,Z 598.905,A -85,B 0,C 180,E1 -17690.584,E2 -17690.584} C_VEL
LIN {X 0,Y 313.644,Z 615.674,A -85,B 0,C 180,E1 -17691.447,E2 -17691.447} C_VEL
LIN {X 0,Y 308.227,Z 633.359,A -85,B 0,C 180,E1 -17692.619,E2 -17692.619} C_VEL
LIN {X 0,Y 302.262,Z 650.275,A -85,B 0,C 180,E1 -17694.047,E2 -17694.047} C_VEL
LIN {X 0,Y 296.765,Z 664.415,A -85,B 0,C 180,E1 -17695.567,E2 -17695.567} C_VEL
LIN {X 0,Y 293.811,Z 672.111,A -85,B 0,C 180,E1 -17696.517,E2 -17696.517} C_VEL
LIN {X 0,Y 291.545,Z 686.474,A -85,B 0,C 180,E1 -17697.639,E2 -17697.639} C_VEL
LIN {X 0,Y 288.837,Z 700.642,A -85,B 0,C 180,E1 -17699.066,E2 -17699.066} C_VEL
LIN {X 0,Y 285.795,Z 713.938,A -85,B 0,C 180,E1 -17700.74,E2 -17700.74} C_VEL
LIN {X 0,Y 282.741,Z 726.034,A -85,B 0,C 180,E1 -17702.621,E2 -17702.621} C_VEL
LIN {X 0,Y 279.802,Z 737.065,A -85,B 0,C 180,E1 -17704.72,E2 -17704.72} C_VEL
LIN {X 0,Y 277.295,Z 746.347,A -85,B 0,C 180,E1 -17706.866,E2 -17706.866} C_VEL
LIN {X 0,Y 274.666,Z 755.451,A -85,B 0,C 180,E1 -17709.399,E2 -17709.399} C_VEL
LIN {X 0,Y 272.523,Z 763,A -85,B 0,C 180,E1 -17711.971,E2 -17711.971} C_VEL
LIN {X 0,Y 270.717,Z 770.034,A -85,B 0,C 180,E1 -17714.951,E2 -17714.951} C_VEL
LIN {X 0,Y 269.412,Z 775.558,A -85,B 0,C 180,E1 -17717.952,E2 -17717.952} C_VEL
LIN {X 0,Y 268.702,Z 779.729,A -85,B 0,C 180,E1 -17720.969,E2 -17720.969} C_VEL
LIN {X 0,Y 268.305,Z 782.649,A -85,B 0,C 180,E1 -17723.983,E2 -17723.983} C_VEL
LIN {X 0,Y 268.199,Z 784.386,A -85,B 0,C 180,E1 -17726.994,E2 -17726.994} C_VEL
LIN {X 0,Y 268.194,Z 784.977,A -85,B 0,C 180,E1 -17729.998,E2 -17729.998} C_VEL
LIN {X 0,Y 268.201,Z 784.377,A -85,B 0,C 180,E1 -17733.002,E2 -17733.002} C_VEL
LIN {X 0,Y 268.297,Z 782.628,A -85,B 0,C 180,E1 -17736.012,E2 -17736.012} C_VEL
LIN {X 0,Y 268.669,Z 779.701,A -85,B 0,C 180,E1 -17739.028,E2 -17739.028} C_VEL
LIN {X 0,Y 269.405,Z 775.525,A -85,B 0,C 180,E1 -17742.043,E2 -17742.043} C_VEL
LIN {X 0,Y 270.704,Z 769.985,A -85,B 0,C 180,E1 -17745.045,E2 -17745.045} C_VEL
LIN {X 0,Y 272.499,Z 762.932,A -85,B 0,C 180,E1 -17748.026,E2 -17748.026} C_VEL
LIN {X 0,Y 274.604,Z 755.371,A -85,B 0,C 180,E1 -17750.601,E2 -17750.601} C_VEL
LIN {X 0,Y 277.268,Z 746.254,A -85,B 0,C 180,E1 -17753.131,E2 -17753.131} C_VEL
LIN {X 0,Y 279.704,Z 736.96,A -85,B 0,C 180,E1 -17755.284,E2 -17755.284} C_VEL
LIN {X 0,Y 282.962,Z 724.9,A -85,B 0,C 180,E1 -17757.552,E2 -17757.552} C_VEL
LIN {X 0,Y 286.031,Z 712.573,A -85,B 0,C 180,E1 -17759.431,E2 -17759.431} C_VEL
LIN {X 0,Y 289.049,Z 698.917,A -85,B 0,C 180,E1 -17761.107,E2 -17761.107} C_VEL
LIN {X 0,Y 291.618,Z 685.363,A -85,B 0,C 180,E1 -17762.436,E2 -17762.436} C_VEL
LIN {X 0,Y 293.761,Z 671.811,A -85,B 0,C 180,E1 -17763.484,E2 -17763.484} C_VEL
LIN {X 0,Y 295.598,Z 657.301,A -85,B 0,C 180,E1 -17764.325,E2 -17764.325} C_VEL
LIN {X 0,Y 297.04,Z 641.23,A -85,B 0,C 180,E1 -17764.958,E2 -17764.958} C_VEL
LIN {X 0,Y 301.077,Z 549.197,A -85,B 0,C 180,E1 -17767.115,E2 -17767.115} C_VEL
LIN {X 0,Y 302.421,Z 514.69,A -85,B 0,C 180,E1 -17767.931,E2 -17767.931} C_VEL
LIN {X 0,Y 299.192,Z 483.448,A -85,B 0,C 180,E1 -17769.359,E2 -17769.359} C_VEL
LIN {X 0,Y 297.422,Z 466.532,A -85,B 0,C 180,E1 -17770.203,E2 -17770.203} C_VEL
LIN {X 0,Y 297.432,Z 462.007,A -85,B 0,C 180,E1 -17770.614,E2 -17770.614} C_VEL
LIN {X 0,Y 292.341,Z 445.042,A -85,B 0,C 180,E1 -17773.161,E2 -17773.161} C_VEL
LIN {X 0,Y 287.492,Z 430.101,A -85,B 0,C 180,E1 -17775.592,E2 -17775.592} C_VEL
LIN {X 0,Y 285.328,Z 422.971,A -85,B 0,C 180,E1 -17776.854,E2 -17776.854} C_VEL
LIN {X 0,Y 283.832,Z 419.671,A -85,B 0,C 180,E1 -17777.566,E2 -17777.566} C_VEL
LIN {X 0,Y 279.178,Z 412.054,A -85,B 0,C 180,E1 -17779.592,E2 -17779.592} C_VEL
LIN {X 0,Y 276.848,Z 408.737,A -85,B 0,C 180,E1 -17780.607,E2 -17780.607} C_VEL
LIN {X 0,Y 276.218,Z 407.309,A -85,B 0,C 180,E1 -17780.954,E2 -17780.954} C_VEL
LIN {X 0,Y 273.963,Z 404.261,A -85,B 0,C 180,E1 -17781.999,E2 -17781.999} C_VEL
LIN {X 0,Y 272.651,Z 401.961,A -85,B 0,C 180,E1 -17782.717,E2 -17782.717} C_VEL
LIN {X 0,Y 271.085,Z 400.071,A -85,B 0,C 180,E1 -17783.479,E2 -17783.479} C_VEL
LIN {X 0,Y 270.294,Z 397.814,A -85,B 0,C 180,E1 -17784.186,E2 -17784.186} C_VEL
LIN {X 0,Y 270.188,Z 397.395,A -85,B 0,C 180,E1 -17784.786,E2 -17784.786} C_VEL
LIN {X 0,Y 270.156,Z 397.46,A -85,B 0,C 180,E1 -17788.648,E2 -17788.648} C_VEL
LIN {X 0,Y 270.184,Z 397.445,A -85,B 0,C 180,E1 -17792.172,E2 -17792.172} C_VEL
LIN {X 0,Y 270.168,Z 397.435,A -85,B 0,C 180,E1 -17795.563,E2 -17795.563} C_VEL
LIN {X 0,Y 270.206,Z 397.429,A -85,B 0,C 180,E1 -17800.237,E2 -17800.237} C_VEL
LIN {X 0,Y 270.324,Z 397.413,A -85,B 0,C 180,E1 -17804.931,E2 -17804.931} C_VEL
LIN {X 0,Y 270.394,Z 397.407,A -85,B 0,C 180,E1 -17809.517,E2 -17809.517} C_VEL
LIN {X 0,Y 270.546,Z 397.404,A -85,B 0,C 180,E1 -17812.537,E2 -17812.537} C_VEL
LIN {X 0,Y 270.756,Z 397.384,A -85,B 0,C 180,E1 -17818.513,E2 -17818.513} C_VEL
LIN {X 0,Y 270.762,Z 397.357,A -85,B 0,C 180,E1 -17821.488,E2 -17821.488} C_VEL
LIN {X 0,Y 270.556,Z 397.386,A -85,B 0,C 180,E1 -17827.463,E2 -17827.463} C_VEL
LIN {X 0,Y 270.374,Z 397.413,A -85,B 0,C 180,E1 -17830.484,E2 -17830.484} C_VEL
LIN {X 0,Y 270.354,Z 397.422,A -85,B 0,C 180,E1 -17835.068,E2 -17835.068} C_VEL
LIN {X 0,Y 270.21,Z 397.441,A -85,B 0,C 180,E1 -17839.763,E2 -17839.763} C_VEL
LIN {X 0,Y 270.171,Z 397.444,A -85,B 0,C 180,E1 -17844.438,E2 -17844.438} C_VEL
LIN {X 0,Y 270.18,Z 397.566,A -85,B 0,C 180,E1 -17848.872,E2 -17848.872} C_VEL
LIN {X 0,Y 270.38,Z 398.602,A -85,B 0,C 180,E1 -17849.381,E2 -17849.381} C_VEL
LIN {X 0,Y 274.561,Z 406.374,A -85,B 0,C 180,E1 -17852.517,E2 -17852.517} C_VEL
LIN {X 0,Y 277.74,Z 412.874,A -85,B 0,C 180,E1 -17854.824,E2 -17854.824} C_VEL
LIN {X 0,Y 282.102,Z 422.917,A -85,B 0,C 180,E1 -17858.068,E2 -17858.068} C_VEL
LIN {X 0,Y 285.729,Z 431.917,A -85,B 0,C 180,E1 -17860.678,E2 -17860.678} C_VEL
LIN {X 0,Y 289.828,Z 443.442,A -85,B 0,C 180,E1 -17863.716,E2 -17863.716} C_VEL
LIN {X 0,Y 293.804,Z 456.924,A -85,B 0,C 180,E1 -17866.851,E2 -17866.851} C_VEL
LIN {X 0,Y 296.493,Z 467.881,A -85,B 0,C 180,E1 -17869.16,E2 -17869.16} C_VEL
LIN {X 0,Y 296.272,Z 471.059,A -85,B 0,C 180,E1 -17869.557,E2 -17869.557} C_VEL
LIN {X 0,Y 301.094,Z 505.03,A -85,B 0,C 180,E1 -17871.36,E2 -17871.36} C_VEL
LIN {X 0,Y 302.859,Z 519.242,A -85,B 0,C 180,E1 -17872.046,E2 -17872.046} C_VEL
LIN {X 0,Y 298.913,Z 614.139,A -85,B 0,C 180,E1 -17874.262,E2 -17874.262} C_VEL
LIN {X 0,Y 297.546,Z 642.383,A -85,B 0,C 180,E1 -17874.955,E2 -17874.955} C_VEL
LIN {X 0,Y 296.219,Z 657.206,A -85,B 0,C 180,E1 -17875.552,E2 -17875.552} C_VEL
LIN {X 0,Y 294.276,Z 671.79,A -85,B 0,C 180,E1 -17876.377,E2 -17876.377} C_VEL
LIN {X 0,Y 291.972,Z 686.209,A -85,B 0,C 180,E1 -17877.486,E2 -17877.486} C_VEL
LIN {X 0,Y 289.574,Z 699.051,A -85,B 0,C 180,E1 -17878.753,E2 -17878.753} C_VEL
LIN {X 0,Y 286.767,Z 711.499,A -85,B 0,C 180,E1 -17880.249,E2 -17880.249} C_VEL
LIN {X 0,Y 283.895,Z 723.057,A -85,B 0,C 180,E1 -17881.945,E2 -17881.945} C_VEL
LIN {X 0,Y 281.295,Z 733.093,A -85,B 0,C 180,E1 -17883.717,E2 -17883.717} C_VEL
LIN {X 0,Y 278.663,Z 743.014,A -85,B 0,C 180,E1 -17885.819,E2 -17885.819} C_VEL
LIN {X 0,Y 275.744,Z 752.794,A -85,B 0,C 180,E1 -17888.314,E2 -17888.314} C_VEL
LIN {X 0,Y 273.432,Z 760.943,A -85,B 0,C 180,E1 -17890.873,E2 -17890.873} C_VEL
LIN {X 0,Y 271.631,Z 767.695,A -85,B 0,C 180,E1 -17893.467,E2 -17893.467} C_VEL
LIN {X 0,Y 270.052,Z 773.954,A -85,B 0,C 180,E1 -17896.457,E2 -17896.457} C_VEL
LIN {X 0,Y 268.973,Z 778.79,A -85,B 0,C 180,E1 -17899.464,E2 -17899.464} C_VEL
LIN {X 0,Y 268.365,Z 782.333,A -85,B 0,C 180,E1 -17902.478,E2 -17902.478} C_VEL
LIN {X 0,Y 268.104,Z 784.674,A -85,B 0,C 180,E1 -17905.492,E2 -17905.492} C_VEL
LIN {X 0,Y 268.125,Z 785.865,A -85,B 0,C 180,E1 -17908.5,E2 -17908.5} C_VEL
LIN {X 0,Y 268.126,Z 785.877,A -85,B 0,C 180,E1 -17911.504,E2 -17911.504} C_VEL
LIN {X 0,Y 268.109,Z 784.737,A -85,B 0,C 180,E1 -17914.513,E2 -17914.513} C_VEL
LIN {X 0,Y 268.369,Z 782.444,A -85,B 0,C 180,E1 -17917.526,E2 -17917.526} C_VEL
LIN {X 0,Y 268.963,Z 778.944,A -85,B 0,C 180,E1 -17920.542,E2 -17920.542} C_VEL
LIN {X 0,Y 270.022,Z 774.158,A -85,B 0,C 180,E1 -17923.549,E2 -17923.549} C_VEL
LIN {X 0,Y 271.551,Z 767.962,A -85,B 0,C 180,E1 -17926.542,E2 -17926.542} C_VEL
LIN {X 0,Y 273.662,Z 760.168,A -85,B 0,C 180,E1 -17929.505,E2 -17929.505} C_VEL
LIN {X 0,Y 276.017,Z 751.853,A -85,B 0,C 180,E1 -17932.062,E2 -17932.062} C_VEL
LIN {X 0,Y 278.795,Z 742.378,A -85,B 0,C 180,E1 -17934.447,E2 -17934.447} C_VEL
LIN {X 0,Y 281.694,Z 731.602,A -85,B 0,C 180,E1 -17936.687,E2 -17936.687} C_VEL
LIN {X 0,Y 284.889,Z 719.337,A -85,B 0,C 180,E1 -17938.756,E2 -17938.756} C_VEL
LIN {X 0,Y 287.835,Z 707.066,A -85,B 0,C 180,E1 -17940.443,E2 -17940.443} C_VEL
LIN {X 0,Y 290.728,Z 693.659,A -85,B 0,C 180,E1 -17941.927,E2 -17941.927} C_VEL
LIN {X 0,Y 293.168,Z 679.608,A -85,B 0,C 180,E1 -17943.173,E2 -17943.173} C_VEL
LIN {X 0,Y 295.224,Z 665.638,A -85,B 0,C 180,E1 -17944.122,E2 -17944.122} C_VEL
LIN {X 0,Y 296.975,Z 650.374,A -85,B 0,C 180,E1 -17944.868,E2 -17944.868} C_VEL
LIN {X 0,Y 298.078,Z 634.189,A -85,B 0,C 180,E1 -17945.391,E2 -17945.391} C_VEL
LIN {X 0,Y 302.344,Z 534.373,A -85,B 0,C 180,E1 -17947.708,E2 -17947.708} C_VEL
LIN {X 0,Y 302.955,Z 519.344,A -85,B 0,C 180,E1 -17948.062,E2 -17948.062} C_VEL
LIN {X 0,Y 298.947,Z 488.671,A -85,B 0,C 180,E1 -17949.593,E2 -17949.593} C_VEL
LIN {X 0,Y 296.332,Z 470.32,A -85,B 0,C 180,E1 -17950.63,E2 -17950.63} C_VEL
LIN {X 0,Y 296.538,Z 467.752,A -85,B 0,C 180,E1 -17950.991,E2 -17950.991} C_VEL
LIN {X 0,Y 293.87,Z 456.969,A -85,B 0,C 180,E1 -17953.26,E2 -17953.26} C_VEL
LIN {X 0,Y 292.258,Z 453.585,A -85,B 0,C 180,E1 -17954.152,E2 -17954.152} C_VEL
LIN {X 0,Y 288.195,Z 449.173,A -85,B 0,C 180,E1 -17955.711,E2 -17955.711} C_VEL
LIN {X 0,Y 284.832,Z 445.846,A -85,B 0,C 180,E1 -17957.003,E2 -17957.003} C_VEL
LIN {X 0,Y 282.822,Z 442.924,A -85,B 0,C 180,E1 -17957.973,E2 -17957.973} C_VEL
LIN {X 0,Y 282.346,Z 441.803,A -85,B 0,C 180,E1 -17958.292,E2 -17958.292} C_VEL
LIN {X 0,Y 278.194,Z 430.325,A -85,B 0,C 180,E1 -17961.553,E2 -17961.553} C_VEL
LIN {X 0,Y 273.413,Z 419.058,A -85,B 0,C 180,E1 -17965.16,E2 -17965.16} C_VEL
LIN {X 0,Y 270.216,Z 412.475,A -85,B 0,C 180,E1 -17967.556,E2 -17967.556} C_VEL
LIN {X 0,Y 269.809,Z 412.083,A -85,B 0,C 180,E1 -17967.778,E2 -17967.778} C_VEL
LIN {X 0,Y 268.865,Z 412.554,A -85,B 0,C 180,E1 -17968.17,E2 -17968.17} C_VEL
LIN {X 0,Y 269.012,Z 413.697,A -85,B 0,C 180,E1 -17968.409,E2 -17968.409} C_VEL
LIN {X 0,Y 278.42,Z 438.709,A -85,B 0,C 180,E1 -17970.225,E2 -17970.225} C_VEL
LIN {X 0,Y 273.103,Z 541.336,A -85,B 0,C 180,E1 -17974.21,E2 -17974.21} C_VEL
LIN {X 0,Y 272.452,Z 557.457,A -85,B 0,C 180,E1 -17975.066,E2 -17975.066} C_VEL
LIN {X 0,Y 271.543,Z 572.405,A -85,B 0,C 180,E1 -17976.146,E2 -17976.146} C_VEL
LIN {X 0,Y 270.418,Z 586.607,A -85,B 0,C 180,E1 -17977.459,E2 -17977.459} C_VEL
LIN {X 0,Y 269.183,Z 601.346,A -85,B 0,C 180,E1 -17979.162,E2 -17979.162} C_VEL
LIN {X 0,Y 267.844,Z 614.388,A -85,B 0,C 180,E1 -17980.999,E2 -17980.999} C_VEL
LIN {X 0,Y 266.679,Z 626.872,A -85,B 0,C 180,E1 -17983.148,E2 -17983.148} C_VEL
LIN {X 0,Y 265.572,Z 637.96,A -85,B 0,C 180,E1 -17985.439,E2 -17985.439} C_VEL
LIN {X 0,Y 264.763,Z 647.227,A -85,B 0,C 180,E1 -17987.739,E2 -17987.739} C_VEL
LIN {X 0,Y 264.127,Z 655.549,A -85,B 0,C 180,E1 -17990.212,E2 -17990.212} C_VEL
LIN {X 0,Y 263.731,Z 661.592,A -85,B 0,C 180,E1 -17992.343,E2 -17992.343} C_VEL
LIN {X 0,Y 263.353,Z 668.7,A -85,B 0,C 180,E1 -17995.408,E2 -17995.408} C_VEL
LIN {X 0,Y 263.609,Z 674.141,A -85,B 0,C 180,E1 -17998.472,E2 -17998.472} C_VEL
LIN {X 0,Y 263.643,Z 676.277,A -85,B 0,C 180,E1 -18000,E2 -18000} C_VEL
LIN {X 0,Y 264.142,Z 678.006,A -85,B 0,C 180,E1 -18001.524,E2 -18001.524} C_VEL
LIN {X 0,Y 265.123,Z 680.434,A -85,B 0,C 180,E1 -18004.561,E2 -18004.561} C_VEL
LIN {X 0,Y 266.443,Z 681.512,A -85,B 0,C 180,E1 -18007.578,E2 -18007.578} C_VEL
LIN {X 0,Y 268.373,Z 681.207,A -85,B 0,C 180,E1 -18010.563,E2 -18010.563} C_VEL
LIN {X 0,Y 270.809,Z 679.547,A -85,B 0,C 180,E1 -18013.507,E2 -18013.507} C_VEL
LIN {X 0,Y 273.948,Z 676.491,A -85,B 0,C 180,E1 -18016.391,E2 -18016.391} C_VEL
LIN {X 0,Y 277.502,Z 672.005,A -85,B 0,C 180,E1 -18019.222,E2 -18019.222} C_VEL
LIN {X 0,Y 281.717,Z 665.966,A -85,B 0,C 180,E1 -18021.975,E2 -18021.975} C_VEL
LIN {X 0,Y 286.425,Z 658.206,A -85,B 0,C 180,E1 -18024.653,E2 -18024.653} C_VEL
LIN {X 0,Y 291.05,Z 649.844,A -85,B 0,C 180,E1 -18026.921,E2 -18026.921} C_VEL
LIN {X 0,Y 296.053,Z 639.841,A -85,B 0,C 180,E1 -18029.12,E2 -18029.12} C_VEL
LIN {X 0,Y 300.647,Z 629.612,A -85,B 0,C 180,E1 -18030.949,E2 -18030.949} C_VEL
LIN {X 0,Y 305.532,Z 617.484,A -85,B 0,C 180,E1 -18032.722,E2 -18032.722} C_VEL
LIN {X 0,Y 309.906,Z 605.455,A -85,B 0,C 180,E1 -18034.144,E2 -18034.144} C_VEL
LIN {X 0,Y 314.436,Z 591.09,A -85,B 0,C 180,E1 -18035.53,E2 -18035.53} C_VEL
LIN {X 0,Y 318.184,Z 576.83,A -85,B 0,C 180,E1 -18036.61,E2 -18036.61} C_VEL
LIN {X 0,Y 322.127,Z 558.482,A -85,B 0,C 180,E1 -18037.691,E2 -18037.691} C_VEL
LIN {X 0,Y 331.152,Z 519.378,A -85,B 0,C 180,E1 -18039.459,E2 -18039.459} C_VEL
LIN {X 0,Y 335.934,Z 499.754,A -85,B 0,C 180,E1 -18040.257,E2 -18040.257} C_VEL
LIN {X 0,Y 335.237,Z 499.857,A -85,B 0,C 180,E1 -18042.133,E2 -18042.133} C_VEL
LIN {X 0,Y 335.06,Z 501.349,A -85,B 0,C 180,E1 -18043.674,E2 -18043.674} C_VEL
LIN {X 0,Y 335.07,Z 503.275,A -85,B 0,C 180,E1 -18044.694,E2 -18044.694} C_VEL
LIN {X 0,Y 332.844,Z 514.597,A -85,B 0,C 180,E1 -18045.691,E2 -18045.691} C_VEL
LIN {X 0,Y 330.993,Z 524.154,A -85,B 0,C 180,E1 -18046.367,E2 -18046.367} C_VEL
LIN {X 0,Y 315.591,Z 596.76,A -85,B 0,C 180,E1 -18049.3,E2 -18049.3} C_VEL
LIN {X 0,Y 311.096,Z 613.37,A -85,B 0,C 180,E1 -18050.129,E2 -18050.129} C_VEL
LIN {X 0,Y 305.167,Z 631.661,A -85,B 0,C 180,E1 -18051.339,E2 -18051.339} C_VEL
LIN {X 0,Y 298.89,Z 648.363,A -85,B 0,C 180,E1 -18052.735,E2 -18052.735} C_VEL
LIN {X 0,Y 292.589,Z 663.524,A -85,B 0,C 180,E1 -18054.372,E2 -18054.372} C_VEL
LIN {X 0,Y 287.411,Z 675.484,A -85,B 0,C 180,E1 -18055.968,E2 -18055.968} C_VEL
LIN {X 0,Y 285.05,Z 689.355,A -85,B 0,C 180,E1 -18057.15,E2 -18057.15} C_VEL
LIN {X 0,Y 282.066,Z 703.497,A -85,B 0,C 180,E1 -18058.657,E2 -18058.657} C_VEL
LIN {X 0,Y 279.031,Z 716.293,A -85,B 0,C 180,E1 -18060.374,E2 -18060.374} C_VEL
LIN {X 0,Y 275.882,Z 727.996,A -85,B 0,C 180,E1 -18062.293,E2 -18062.293} C_VEL
LIN {X 0,Y 272.675,Z 739.307,A -85,B 0,C 180,E1 -18064.574,E2 -18064.574} C_VEL
LIN {X 0,Y 269.839,Z 749.114,A -85,B 0,C 180,E1 -18067.001,E2 -18067.001} C_VEL
LIN {X 0,Y 267.301,Z 757.756,A -85,B 0,C 180,E1 -18069.61,E2 -18069.61} C_VEL
LIN {X 0,Y 265.178,Z 764.939,A -85,B 0,C 180,E1 -18072.253,E2 -18072.253} C_VEL
LIN {X 0,Y 263.452,Z 771.574,A -85,B 0,C 180,E1 -18075.317,E2 -18075.317} C_VEL
LIN {X 0,Y 262.21,Z 776.76,A -85,B 0,C 180,E1 -18078.401,E2 -18078.401} C_VEL
LIN {X 0,Y 261.664,Z 779.744,A -85,B 0,C 180,E1 -18080.724,E2 -18080.724} C_VEL
LIN {X 0,Y 261.231,Z 782.664,A -85,B 0,C 180,E1 -18083.82,E2 -18083.82} C_VEL
LIN {X 0,Y 261.094,Z 784.401,A -85,B 0,C 180,E1 -18086.912,E2 -18086.912} C_VEL
LIN {X 0,Y 261.121,Z 784.99,A -85,B 0,C 180,E1 -18089.998,E2 -18089.998} C_VEL
LIN {X 0,Y 261.096,Z 784.391,A -85,B 0,C 180,E1 -18093.084,E2 -18093.084} C_VEL
LIN {X 0,Y 261.224,Z 782.641,A -85,B 0,C 180,E1 -18096.175,E2 -18096.175} C_VEL
LIN {X 0,Y 261.637,Z 779.715,A -85,B 0,C 180,E1 -18099.272,E2 -18099.272} C_VEL
LIN {X 0,Y 262.412,Z 775.539,A -85,B 0,C 180,E1 -18102.369,E2 -18102.369} C_VEL
LIN {X 0,Y 263.785,Z 770,A -85,B 0,C 180,E1 -18105.449,E2 -18105.449} C_VEL
LIN {X 0,Y 265.695,Z 762.947,A -85,B 0,C 180,E1 -18108.504,E2 -18108.504} C_VEL
LIN {X 0,Y 267.92,Z 755.386,A -85,B 0,C 180,E1 -18111.14,E2 -18111.14} C_VEL
LIN {X 0,Y 270.719,Z 746.27,A -85,B 0,C 180,E1 -18113.725,E2 -18113.725} C_VEL
LIN {X 0,Y 273.26,Z 736.977,A -85,B 0,C 180,E1 -18115.924,E2 -18115.924} C_VEL
LIN {X 0,Y 276.662,Z 724.919,A -85,B 0,C 180,E1 -18118.235,E2 -18118.235} C_VEL
LIN {X 0,Y 279.86,Z 712.595,A -85,B 0,C 180,E1 -18120.146,E2 -18120.146} C_VEL
LIN {X 0,Y 282.97,Z 698.942,A -85,B 0,C 180,E1 -18121.852,E2 -18121.852} C_VEL
LIN {X 0,Y 285.744,Z 684.773,A -85,B 0,C 180,E1 -18123.255,E2 -18123.255} C_VEL
LIN {X 0,Y 288.05,Z 670.575,A -85,B 0,C 180,E1 -18124.345,E2 -18124.345} C_VEL
LIN {X 0,Y 289.909,Z 656.49,A -85,B 0,C 180,E1 -18125.149,E2 -18125.149} C_VEL
LIN {X 0,Y 291.26,Z 641.313,A -85,B 0,C 180,E1 -18125.757,E2 -18125.757} C_VEL
LIN {X 0,Y 295.412,Z 550.024,A -85,B 0,C 180,E1 -18127.93,E2 -18127.93} C_VEL
LIN {X 0,Y 296.83,Z 515.552,A -85,B 0,C 180,E1 -18128.755,E2 -18128.755} C_VEL
LIN {X 0,Y 293.471,Z 481.92,A -85,B 0,C 180,E1 -18130.334,E2 -18130.334} C_VEL
LIN {X 0,Y 291.869,Z 467.471,A -85,B 0,C 180,E1 -18131.063,E2 -18131.063} C_VEL
LIN {X 0,Y 291.641,Z 464.12,A -85,B 0,C 180,E1 -18131.405,E2 -18131.405} C_VEL
LIN {X 0,Y 286.692,Z 447.203,A -85,B 0,C 180,E1 -18134.039,E2 -18134.039} C_VEL
LIN {X 0,Y 281.26,Z 429.348,A -85,B 0,C 180,E1 -18137.085,E2 -18137.085} C_VEL
LIN {X 0,Y 279.592,Z 424.96,A -85,B 0,C 180,E1 -18137.987,E2 -18137.987} C_VEL
LIN {X 0,Y 274.599,Z 416.879,A -85,B 0,C 180,E1 -18140.22,E2 -18140.22} C_VEL
LIN {X 0,Y 268.953,Z 407.803,A -85,B 0,C 180,E1 -18143.058,E2 -18143.058} C_VEL
LIN {X 0,Y 267.096,Z 405.376,A -85,B 0,C 180,E1 -18144.015,E2 -18144.015} C_VEL
LIN {X 0,Y 266.369,Z 403.639,A -85,B 0,C 180,E1 -18144.517,E2 -18144.517} C_VEL
LIN {X 0,Y 264.58,Z 401.753,A -85,B 0,C 180,E1 -18145.426,E2 -18145.426} C_VEL
LIN {X 0,Y 263.247,Z 398.806,A -85,B 0,C 180,E1 -18146.475,E2 -18146.475} C_VEL
LIN {X 0,Y 263.139,Z 398.313,A -85,B 0,C 180,E1 -18147.031,E2 -18147.031} C_VEL
LIN {X 0,Y 263.129,Z 398.319,A -85,B 0,C 180,E1 -18151.806,E2 -18151.806} C_VEL
LIN {X 0,Y 263.101,Z 398.321,A -85,B 0,C 180,E1 -18156.379,E2 -18156.379} C_VEL
LIN {X 0,Y 263.194,Z 398.303,A -85,B 0,C 180,E1 -18159.688,E2 -18159.688} C_VEL
LIN {X 0,Y 263.274,Z 398.292,A -85,B 0,C 180,E1 -18164.518,E2 -18164.518} C_VEL
LIN {X 0,Y 263.333,Z 398.289,A -85,B 0,C 180,E1 -18169.233,E2 -18169.233} C_VEL
LIN {X 0,Y 263.51,Z 398.277,A -85,B 0,C 180,E1 -18172.337,E2 -18172.337} C_VEL
LIN {X 0,Y 263.719,Z 398.26,A -85,B 0,C 180,E1 -18178.473,E2 -18178.473} C_VEL
LIN {X 0,Y 263.725,Z 398.233,A -85,B 0,C 180,E1 -18181.527,E2 -18181.527} C_VEL
LIN {X 0,Y 263.518,Z 398.264,A -85,B 0,C 180,E1 -18187.663,E2 -18187.663} C_VEL
LIN {X 0,Y 263.32,Z 398.288,A -85,B 0,C 180,E1 -18190.768,E2 -18190.768} C_VEL
LIN {X 0,Y 263.297,Z 398.294,A -85,B 0,C 180,E1 -18195.481,E2 -18195.481} C_VEL
LIN {X 0,Y 263.195,Z 398.308,A -85,B 0,C 180,E1 -18200.312,E2 -18200.312} C_VEL
LIN {X 0,Y 263.108,Z 398.318,A -85,B 0,C 180,E1 -18205.302,E2 -18205.302} C_VEL
LIN {X 0,Y 263.138,Z 398.58,A -85,B 0,C 180,E1 -18206.735,E2 -18206.735} C_VEL
LIN {X 0,Y 264.178,Z 401.244,A -85,B 0,C 180,E1 -18207.923,E2 -18207.923} C_VEL
LIN {X 0,Y 265.038,Z 402.356,A -85,B 0,C 180,E1 -18208.51,E2 -18208.51} C_VEL
LIN {X 0,Y 269.791,Z 411.663,A -85,B 0,C 180,E1 -18212.345,E2 -18212.345} C_VEL
LIN {X 0,Y 273.737,Z 419.952,A -85,B 0,C 180,E1 -18215.287,E2 -18215.287} C_VEL
LIN {X 0,Y 278.18,Z 430.484,A -85,B 0,C 180,E1 -18218.658,E2 -18218.658} C_VEL
LIN {X 0,Y 282.07,Z 440.979,A -85,B 0,C 180,E1 -18221.632,E2 -18221.632} C_VEL
LIN {X 0,Y 284.741,Z 448.99,A -85,B 0,C 180,E1 -18223.717,E2 -18223.717} C_VEL
LIN {X 0,Y 288.388,Z 461.681,A -85,B 0,C 180,E1 -18226.697,E2 -18226.697} C_VEL
LIN {X 0,Y 290.587,Z 470.587,A -85,B 0,C 180,E1 -18228.569,E2 -18228.569} C_VEL
LIN {X 0,Y 293.854,Z 493.359,A -85,B 0,C 180,E1 -18229.862,E2 -18229.862} C_VEL
LIN {X 0,Y 297.258,Z 520.294,A -85,B 0,C 180,E1 -18231.234,E2 -18231.234} C_VEL
LIN {X 0,Y 293.005,Z 617.605,A -85,B 0,C 180,E1 -18233.533,E2 -18233.533} C_VEL
LIN {X 0,Y 291.67,Z 643.603,A -85,B 0,C 180,E1 -18234.195,E2 -18234.195} C_VEL
LIN {X 0,Y 290.212,Z 658.835,A -85,B 0,C 180,E1 -18234.84,E2 -18234.84} C_VEL
LIN {X 0,Y 288.046,Z 674.145,A -85,B 0,C 180,E1 -18235.76,E2 -18235.76} C_VEL
LIN {X 0,Y 285.615,Z 688.306,A -85,B 0,C 180,E1 -18236.91,E2 -18236.91} C_VEL
LIN {X 0,Y 282.878,Z 702.052,A -85,B 0,C 180,E1 -18238.345,E2 -18238.345} C_VEL
LIN {X 0,Y 279.643,Z 715.202,A -85,B 0,C 180,E1 -18240.036,E2 -18240.036} C_VEL
LIN {X 0,Y 276.468,Z 727.188,A -85,B 0,C 180,E1 -18241.95,E2 -18241.95} C_VEL
LIN {X 0,Y 273.456,Z 738.142,A -85,B 0,C 180,E1 -18244.096,E2 -18244.096} C_VEL
LIN {X 0,Y 270.817,Z 747.372,A -85,B 0,C 180,E1 -18246.284,E2 -18246.284} C_VEL
LIN {X 0,Y 268.014,Z 756.438,A -85,B 0,C 180,E1 -18248.868,E2 -18248.868} C_VEL
LIN {X 0,Y 265.782,Z 763.967,A -85,B 0,C 180,E1 -18251.502,E2 -18251.502} C_VEL
LIN {X 0,Y 263.852,Z 770.998,A -85,B 0,C 180,E1 -18254.555,E2 -18254.555} C_VEL
LIN {X 0,Y 262.406,Z 776.527,A -85,B 0,C 180,E1 -18257.63,E2 -18257.63} C_VEL
LIN {X 0,Y 261.581,Z 780.703,A -85,B 0,C 180,E1 -18260.726,E2 -18260.726} C_VEL
LIN {X 0,Y 261.142,Z 783.636,A -85,B 0,C 180,E1 -18263.823,E2 -18263.823} C_VEL
LIN {X 0,Y 260.999,Z 785.398,A -85,B 0,C 180,E1 -18266.915,E2 -18266.915} C_VEL
LIN {X 0,Y 261.035,Z 786.008,A -85,B 0,C 180,E1 -18270.002,E2 -18270.002} C_VEL
LIN {X 0,Y 261.002,Z 785.435,A -85,B 0,C 180,E1 -18273.089,E2 -18273.089} C_VEL
LIN {X 0,Y 261.147,Z 783.723,A -85,B 0,C 180,E1 -18276.182,E2 -18276.182} C_VEL
LIN {X 0,Y 261.582,Z 780.834,A -85,B 0,C 180,E1 -18279.279,E2 -18279.279} C_VEL
LIN {X 0,Y 262.383,Z 776.703,A -85,B 0,C 180,E1 -18282.376,E2 -18282.376} C_VEL
LIN {X 0,Y 263.804,Z 771.229,A -85,B 0,C 180,E1 -18285.453,E2 -18285.453} C_VEL
LIN {X 0,Y 265.7,Z 764.262,A -85,B 0,C 180,E1 -18288.509,E2 -18288.509} C_VEL
LIN {X 0,Y 267.929,Z 756.792,A -85,B 0,C 180,E1 -18291.144,E2 -18291.144} C_VEL
LIN {X 0,Y 270.732,Z 747.793,A -85,B 0,C 180,E1 -18293.728,E2 -18293.728} C_VEL
LIN {X 0,Y 273.832,Z 736.916,A -85,B 0,C 180,E1 -18296.28,E2 -18296.28} C_VEL
LIN {X 0,Y 276.991,Z 725.736,A -85,B 0,C 180,E1 -18298.41,E2 -18298.41} C_VEL
LIN {X 0,Y 280.139,Z 713.458,A -85,B 0,C 180,E1 -18300.326,E2 -18300.326} C_VEL
LIN {X 0,Y 283.383,Z 699.909,A -85,B 0,C 180,E1 -18302.015,E2 -18302.015} C_VEL
LIN {X 0,Y 286.129,Z 685.956,A -85,B 0,C 180,E1 -18303.412,E2 -18303.412} C_VEL
LIN {X 0,Y 288.436,Z 671.907,A -85,B 0,C 180,E1 -18304.509,E2 -18304.509} C_VEL
LIN {X 0,Y 290.431,Z 657.365,A -85,B 0,C 180,E1 -18305.347,E2 -18305.347} C_VEL
LIN {X 0,Y 291.847,Z 642.656,A -85,B 0,C 180,E1 -18305.945,E2 -18305.945} C_VEL
LIN {X 0,Y 293.442,Z 609.138,A -85,B 0,C 180,E1 -18306.783,E2 -18306.783} C_VEL
LIN {X 0,Y 297.41,Z 521.161,A -85,B 0,C 180,E1 -18308.843,E2 -18308.843} C_VEL
LIN {X 0,Y 293.55,Z 490.592,A -85,B 0,C 180,E1 -18310.405,E2 -18310.405} C_VEL
LIN {X 0,Y 290.604,Z 470.572,A -85,B 0,C 180,E1 -18311.566,E2 -18311.566} C_VEL
LIN {X 0,Y 287.854,Z 459.753,A -85,B 0,C 180,E1 -18313.84,E2 -18313.84} C_VEL
LIN {X 0,Y 284.907,Z 449.459,A -85,B 0,C 180,E1 -18316.315,E2 -18316.315} C_VEL
LIN {X 0,Y 282.346,Z 441.803,A -85,B 0,C 180,E1 -18318.292,E2 -18318.292} C_VEL
LIN {X 0,Y 280.64,Z 438.794,A -85,B 0,C 180,E1 -18319.266,E2 -18319.266} C_VEL
LIN {X 0,Y 276.558,Z 435.152,A -85,B 0,C 180,E1 -18320.968,E2 -18320.968} C_VEL
LIN {X 0,Y 273.162,Z 432.462,A -85,B 0,C 180,E1 -18322.374,E2 -18322.374} C_VEL
LIN {X 0,Y 271.107,Z 429.967,A -85,B 0,C 180,E1 -18323.433,E2 -18323.433} C_VEL
LIN {X 0,Y 270.59,Z 428.968,A -85,B 0,C 180,E1 -18323.781,E2 -18323.781} C_VEL
LIN {X 0,Y 267.177,Z 421.076,A -85,B 0,C 180,E1 -18326.468,E2 -18326.468} C_VEL
LIN {X 0,Y 265.704,Z 418.56,A -85,B 0,C 180,E1 -18327.5,E2 -18327.5} C_VEL
LIN {X 0,Y 264.107,Z 419.136,A -85,B 0,C 180,E1 -18328.047,E2 -18328.047} C_VEL
LIN {X 0,Y 264.165,Z 420.15,A -85,B 0,C 180,E1 -18328.308,E2 -18328.308} C_VEL
LIN {X 0,Y 271.685,Z 440.63,A -85,B 0,C 180,E1 -18329.825,E2 -18329.825} C_VEL
LIN {X 0,Y 266.325,Z 538.842,A -85,B 0,C 180,E1 -18333.755,E2 -18333.755} C_VEL
LIN {X 0,Y 265.604,Z 555.351,A -85,B 0,C 180,E1 -18334.599,E2 -18334.599} C_VEL
LIN {X 0,Y 264.702,Z 570.899,A -85,B 0,C 180,E1 -18335.699,E2 -18335.699} C_VEL
LIN {X 0,Y 263.543,Z 585.682,A -85,B 0,C 180,E1 -18337.045,E2 -18337.045} C_VEL
LIN {X 0,Y 262.289,Z 600.758,A -85,B 0,C 180,E1 -18338.793,E2 -18338.793} C_VEL
LIN {X 0,Y 260.87,Z 614.233,A -85,B 0,C 180,E1 -18340.707,E2 -18340.707} C_VEL
LIN {X 0,Y 259.696,Z 626.777,A -85,B 0,C 180,E1 -18342.884,E2 -18342.884} C_VEL
LIN {X 0,Y 258.623,Z 637.149,A -85,B 0,C 180,E1 -18345.039,E2 -18345.039} C_VEL
LIN {X 0,Y 257.791,Z 646.72,A -85,B 0,C 180,E1 -18347.402,E2 -18347.402} C_VEL
LIN {X 0,Y 257.043,Z 655.969,A -85,B 0,C 180,E1 -18350.149,E2 -18350.149} C_VEL
LIN {X 0,Y 256.558,Z 663.631,A -85,B 0,C 180,E1 -18352.919,E2 -18352.919} C_VEL
LIN {X 0,Y 256.282,Z 668.99,A -85,B 0,C 180,E1 -18355.281,E2 -18355.281} C_VEL
LIN {X 0,Y 256.522,Z 674.628,A -85,B 0,C 180,E1 -18358.43,E2 -18358.43} C_VEL
LIN {X 0,Y 256.571,Z 676.899,A -85,B 0,C 180,E1 -18360,E2 -18360} C_VEL
LIN {X 0,Y 257.084,Z 678.772,A -85,B 0,C 180,E1 -18361.566,E2 -18361.566} C_VEL
LIN {X 0,Y 258.138,Z 681.474,A -85,B 0,C 180,E1 -18364.685,E2 -18364.685} C_VEL
LIN {X 0,Y 259.534,Z 682.812,A -85,B 0,C 180,E1 -18367.781,E2 -18367.781} C_VEL
LIN {X 0,Y 261.584,Z 682.748,A -85,B 0,C 180,E1 -18370.84,E2 -18370.84} C_VEL
LIN {X 0,Y 264.155,Z 681.375,A -85,B 0,C 180,E1 -18373.854,E2 -18373.854} C_VEL
LIN {X 0,Y 267.463,Z 678.559,A -85,B 0,C 180,E1 -18376.8,E2 -18376.8} C_VEL
LIN {X 0,Y 271.212,Z 674.4,A -85,B 0,C 180,E1 -18379.686,E2 -18379.686} C_VEL
LIN {X 0,Y 275.63,Z 668.727,A -85,B 0,C 180,E1 -18382.487,E2 -18382.487} C_VEL
LIN {X 0,Y 280.595,Z 661.473,A -85,B 0,C 180,E1 -18385.201,E2 -18385.201} C_VEL
LIN {X 0,Y 285.429,Z 653.581,A -85,B 0,C 180,E1 -18387.495,E2 -18387.495} C_VEL
LIN {X 0,Y 290.668,Z 644.109,A -85,B 0,C 180,E1 -18389.713,E2 -18389.713} C_VEL
LIN {X 0,Y 295.469,Z 634.534,A -85,B 0,C 180,E1 -18391.553,E2 -18391.553} C_VEL
LIN {X 0,Y 301.04,Z 622.281,A -85,B 0,C 180,E1 -18393.473,E2 -18393.473} C_VEL
LIN {X 0,Y 306.094,Z 609.784,A -85,B 0,C 180,E1 -18395.03,E2 -18395.03} C_VEL
LIN {X 0,Y 311.348,Z 594.722,A -85,B 0,C 180,E1 -18396.538,E2 -18396.538} C_VEL
LIN {X 0,Y 315.322,Z 581.315,A -85,B 0,C 180,E1 -18397.6,E2 -18397.6} C_VEL
LIN {X 0,Y 319.21,Z 565.07,A -85,B 0,C 180,E1 -18398.612,E2 -18398.612} C_VEL
LIN {X 0,Y 324.07,Z 544.415,A -85,B 0,C 180,E1 -18399.622,E2 -18399.622} C_VEL
LIN {X 0,Y 333.631,Z 506.453,A -85,B 0,C 180,E1 -18401.232,E2 -18401.232} C_VEL
LIN {X 0,Y 333.243,Z 507.308,A -85,B 0,C 180,E1 -18402.855,E2 -18402.855} C_VEL
LIN {X 0,Y 333.112,Z 508.855,A -85,B 0,C 180,E1 -18403.866,E2 -18403.866} C_VEL
LIN {X 0,Y 330.538,Z 520.488,A -85,B 0,C 180,E1 -18404.851,E2 -18404.851} C_VEL
LIN {X 0,Y 329.29,Z 526.252,A -85,B 0,C 180,E1 -18405.224,E2 -18405.224} C_VEL
LIN {X 0,Y 313.968,Z 593.566,A -85,B 0,C 180,E1 -18407.914,E2 -18407.914} C_VEL
LIN {X 0,Y 308.835,Z 611.623,A -85,B 0,C 180,E1 -18408.811,E2 -18408.811} C_VEL
LIN {X 0,Y 302.926,Z 628.829,A -85,B 0,C 180,E1 -18409.921,E2 -18409.921} C_VEL
LIN {X 0,Y 296.38,Z 645.436,A -85,B 0,C 180,E1 -18411.285,E2 -18411.285} C_VEL
LIN {X 0,Y 290.168,Z 659.518,A -85,B 0,C 180,E1 -18412.732,E2 -18412.732} C_VEL
LIN {X 0,Y 284.04,Z 672.632,A -85,B 0,C 180,E1 -18414.444,E2 -18414.444} C_VEL
LIN {X 0,Y 280.93,Z 679.231,A -85,B 0,C 180,E1 -18415.451,E2 -18415.451} C_VEL
LIN {X 0,Y 278.42,Z 692.884,A -85,B 0,C 180,E1 -18416.698,E2 -18416.698} C_VEL
LIN {X 0,Y 275.381,Z 706.351,A -85,B 0,C 180,E1 -18418.237,E2 -18418.237} C_VEL
LIN {X 0,Y 271.932,Z 719.778,A -85,B 0,C 180,E1 -18420.162,E2 -18420.162} C_VEL
LIN {X 0,Y 268.482,Z 731.836,A -85,B 0,C 180,E1 -18422.311,E2 -18422.311} C_VEL
LIN {X 0,Y 265.582,Z 741.758,A -85,B 0,C 180,E1 -18424.477,E2 -18424.477} C_VEL
LIN {X 0,Y 262.428,Z 751.813,A -85,B 0,C 180,E1 -18427.148,E2 -18427.148} C_VEL
LIN {X 0,Y 259.93,Z 759.995,A -85,B 0,C 180,E1 -18429.832,E2 -18429.832} C_VEL
LIN {X 0,Y 257.781,Z 766.862,A -85,B 0,C 180,E1 -18432.596,E2 -18432.596} C_VEL
LIN {X 0,Y 256.16,Z 773.005,A -85,B 0,C 180,E1 -18435.702,E2 -18435.702} C_VEL
LIN {X 0,Y 254.977,Z 777.836,A -85,B 0,C 180,E1 -18438.873,E2 -18438.873} C_VEL
LIN {X 0,Y 254.334,Z 781.37,A -85,B 0,C 180,E1 -18442.056,E2 -18442.056} C_VEL
LIN {X 0,Y 254.042,Z 783.691,A -85,B 0,C 180,E1 -18445.237,E2 -18445.237} C_VEL
LIN {X 0,Y 254.015,Z 784.853,A -85,B 0,C 180,E1 -18448.412,E2 -18448.412} C_VEL
LIN {X 0,Y 254.018,Z 784.85,A -85,B 0,C 180,E1 -18451.583,E2 -18451.583} C_VEL
LIN {X 0,Y 254.041,Z 783.467,A -85,B 0,C 180,E1 -18455.17,E2 -18455.17} C_VEL
LIN {X 0,Y 254.311,Z 781.342,A -85,B 0,C 180,E1 -18457.94,E2 -18457.94} C_VEL
LIN {X 0,Y 254.965,Z 777.803,A -85,B 0,C 180,E1 -18461.122,E2 -18461.122} C_VEL
LIN {X 0,Y 256.15,Z 772.962,A -85,B 0,C 180,E1 -18464.293,E2 -18464.293} C_VEL
LIN {X 0,Y 257.799,Z 766.688,A -85,B 0,C 180,E1 -18467.447,E2 -18467.447} C_VEL
LIN {X 0,Y 260.199,Z 758.804,A -85,B 0,C 180,E1 -18470.554,E2 -18470.554} C_VEL
LIN {X 0,Y 262.792,Z 750.386,A -85,B 0,C 180,E1 -18473.23,E2 -18473.23} C_VEL
LIN {X 0,Y 265.452,Z 741.893,A -85,B 0,C 180,E1 -18475.465,E2 -18475.465} C_VEL
LIN {X 0,Y 268.465,Z 731.712,A -85,B 0,C 180,E1 -18477.686,E2 -18477.686} C_VEL
LIN {X 0,Y 271.848,Z 719.633,A -85,B 0,C 180,E1 -18479.842,E2 -18479.842} C_VEL
LIN {X 0,Y 275.336,Z 706.153,A -85,B 0,C 180,E1 -18481.763,E2 -18481.763} C_VEL
LIN {X 0,Y 278.329,Z 692.622,A -85,B 0,C 180,E1 -18483.309,E2 -18483.309} C_VEL
LIN {X 0,Y 280.94,Z 678.595,A -85,B 0,C 180,E1 -18484.576,E2 -18484.576} C_VEL
LIN {X 0,Y 283.142,Z 664.136,A -85,B 0,C 180,E1 -18485.571,E2 -18485.571} C_VEL
LIN {X 0,Y 284.901,Z 649.306,A -85,B 0,C 180,E1 -18486.298,E2 -18486.298} C_VEL
LIN {X 0,Y 286.047,Z 634.065,A -85,B 0,C 180,E1 -18486.786,E2 -18486.786} C_VEL
LIN {X 0,Y 289.972,Z 547.537,A -85,B 0,C 180,E1 -18488.853,E2 -18488.853} C_VEL
LIN {X 0,Y 291.322,Z 516.649,A -85,B 0,C 180,E1 -18489.599,E2 -18489.599} C_VEL
LIN {X 0,Y 287.899,Z 481.469,A -85,B 0,C 180,E1 -18491.3,E2 -18491.3} C_VEL
LIN {X 0,Y 286.288,Z 467.526,A -85,B 0,C 180,E1 -18492.046,E2 -18492.046} C_VEL
LIN {X 0,Y 281.267,Z 449.989,A -85,B 0,C 180,E1 -18494.846,E2 -18494.846} C_VEL
LIN {X 0,Y 276.616,Z 433.862,A -85,B 0,C 180,E1 -18497.678,E2 -18497.678} C_VEL
LIN {X 0,Y 275.316,Z 430.222,A -85,B 0,C 180,E1 -18498.417,E2 -18498.417} C_VEL
LIN {X 0,Y 270.069,Z 421.647,A -85,B 0,C 180,E1 -18500.872,E2 -18500.872} C_VEL
LIN {X 0,Y 265.263,Z 413.654,A -85,B 0,C 180,E1 -18503.407,E2 -18503.407} C_VEL
LIN {X 0,Y 262.336,Z 409.089,A -85,B 0,C 180,E1 -18505.088,E2 -18505.088} C_VEL
LIN {X 0,Y 260.114,Z 406.117,A -85,B 0,C 180,E1 -18506.366,E2 -18506.366} C_VEL
LIN {X 0,Y 258.994,Z 404.053,A -85,B 0,C 180,E1 -18507.132,E2 -18507.132} C_VEL
LIN {X 0,Y 257.49,Z 402.626,A -85,B 0,C 180,E1 -18507.965,E2 -18507.965} C_VEL
LIN {X 0,Y 256.142,Z 399.688,A -85,B 0,C 180,E1 -18509.153,E2 -18509.153} C_VEL
LIN {X 0,Y 256.035,Z 399.203,A -85,B 0,C 180,E1 -18509.937,E2 -18509.937} C_VEL
